# B&R Automation Studio project TD52 (part 124)

#### ChCCyclic.st
```iecst
(*******************************************************************************
ChC 			charge cooler

This code is confidential AND proprietary to the INNIO Company.
It may NOT be used in any form, OR reproduced in any manner,
without written permission of the INNIO Company.
Copyright, INNIO Company, 2019

Customized modifications: -
------------------------

History:
-------
V2.30	24.01.2008	LH			erstellt (Kopie von kv_schr)
 		06.02.2008	LH			angepasst an Auto-Tune Regler
V3.10.0	17.02.2010	lettenb.	corr.demand fan stage 1,2  step10: AND NOT FA_PLUS.Q --> AND FA_PLUS.Q
								corr. Anz_GK_anfhbt LIMIT(1->0,...)  	fehlerbehebung(robert mayer)
V3.99.0	21.02.2013	lettenb.	parts from pb3 included
		24.06.2013	lettenb.	xGRMin_Ventpos: Hy:= 1->0.01, bugfix
V4.00.0	03.03.2015	lettenb.	GK_frg (IN_HC.bChC_Rel) moved TO MM_CU
V4.03.0 07.08.2015  Denk		Manual operating auxiliaries control functionality added
        30.09.2015  Plattner	charge cooling pre heating OUT_HC.tChC_Heating.Do added
V4.07.0	09.08.2018	Schmid		2nd low temperature charge cooling circuit added
		08.01.2019	Schmid		redundant pump control
		22.02.2019	Schmid		Charge cooler heating bugfix

Instructions for use:
--------------------

Outstandings:
------------
(*******************************************************************************)
PROGRAM _CYCLIC
	//parameter definitions see settingsInit.st
	(* charge cooler 1st LT cooling circuit *)
	GK_var 			:= INT_TO_USINT(LIMIT(0, Para.iChC_OpMode,    2));		(* cooler mode (0-2)
																			0 = no cooler
																			1 = cooler level dependent on valve position supply water temperature controller
																			2 = cooler level dependent on charge (supply water) temperature *)
	GK_anz			:= INT_TO_USINT(LIMIT(1, Para.iChC_NumStages, 16));		(* number stages total (1-16)*)
	Anz_GK_anfhbt	:= INT_TO_USINT(LIMIT(0, Para.iChC_NumDemAux, GK_anz));	(* number stages with demand auxiliaries (0-16)*)
	GK_reg			:= INT_TO_USINT(LIMIT(1, Para.iChC_CtrNum, 9));			(* number controller for y for 3-way valve (1-9) (mode 1) *)
																			(* 1-8 = Ctr_Cust	plant controller - custom		*)
																			(*   9 = Ctr_ChC	charge temperature (t2') controller	*)

	(* charge cooler 2nd LT cooling circuit *)
	GK2_var 		:= INT_TO_USINT(LIMIT(0, Para.iChC2_OpMode,    22));	 (* cooler 2 fan operation mode (0-22)
																			 0	= LT circuits are connected, cooler fan controlled by 1st circuit (t2'), cooler 2 fan not connected
																			 11	= separate LT circuits, combi-cooler, cooler fan stage control for 2nd circuit dependent
																				  on temperature-control-valve position, cooler 2 fan not connected
																			 12	= separate LT circuits, combi-cooler, cooler fan stage control FOR 2nd circuit dependent
																				  on charge temperature (T1-HP), cooler 2 fan not connected
																			 21 = separate LT circuits, separate cooler fans, stage control dependent
																				  on temperature-control-valve position
																			 22 = separate LT circuits, separate cooler fans, stage control dependent
																				  on charge temperature (T1-HP) *)
	IF GK2_var > 20 THEN	(* separate 2nd charge cooler *)
		GK2_anz			:= INT_TO_USINT(LIMIT(1, Para.iChC2_NumStages, 16));	 	(* number stages total (1-16)*)
		Anz_GK2_anfhbt	:= INT_TO_USINT(LIMIT(0, Para.iChC2_NumDemAux, GK2_anz));	(* number stages with demand auxiliaries (0-16)*)
	ELSE					(* no 2nd charge cooler or combi-cooler *)
		GK2_anz			:= GK_anz;
		Anz_GK2_anfhbt	:= Anz_GK_anfhbt;
	END_IF;
	GK2_reg			:= INT_TO_USINT(LIMIT(1, Para.iChC2_CtrNum, 34));		 (* number controller for y for 3-way valve (1-8, 34)*)
																			 (* 1-8 = Ctr_Cust		plant controller - custom		*)
																			 (*  34 = Ctr_ChC_T1HP	charge temperature before high-pressure turbo charger (T1-HP) controller	*)

	(*------------------------------------------------------------------------------------------*)
	(* charge cooler pump *)
	OUT_HC.tChC_DemPump.Do		:= IN_HC.bEng_Aux_Dem_CDR
								OR IN_HC.tManAuxCtr.bChC_DemPump;	(* Manual operating auxiliaries control - Handbedienebene *)
	OUT_HC.bCCWP_Dem			:= OUT_HC.tChC_DemPump.Do;

	(* charge cooler 2 pump *)
	OUT_HC.tChC2_DemPump.Do		:= IN_HC.bEng_Aux_Dem_CDR
								OR IN_HC.tManAuxCtr.bChC2_DemPump;	(* Manual operating auxiliaries control - Handbedienebene *)
	OUT_HC.bCC2WP_Dem			:= OUT_HC.tChC2_DemPump.Do;

	(* release charge cooler from monitoring (remove not applicable parts) *)
	IN_HC.bChC_Rel;
	IN_HC.bChC2_Rel;

	(*==========================================================================================*)
	(* charge cooler control - stepper version *)
	IF GK_var > 0 THEN
		(* cooler stages ON/OFF according charge cooler mode *)
		(* if necessary change with limit value charge cooler water temperature *)
		bChC_Up   :=     bT_Ch_Hi2;
		bChC_Down := NOT bT_Ch_Hi1;

		(*------------------------------------------------------------------------------------------*)
		IF GK_var > 1 THEN
			Temp_KuehlerAustritt := 1;
		ELSE
			Temp_KuehlerAustritt := 0;
		END_IF;

		GK_vent			:=	0;
		GK_temp			:=	0;
		IF Temp_KuehlerAustritt THEN
			GK_temp		:=	1;
		ELSIF Para.bCtr_ChC THEN
			GK_vent		:=	1;
		END_IF;

		IF	Anz_GK_anfhbt > 0 THEN
			GK_anfhbt	:=	1;
		ELSE
			GK_anfhbt	:=	0;
		END_IF;

		FOR	i:=	1 TO 16 BY 1 DO
			gk_anfhbt[i] :=	0;
		END_FOR;
		FOR	i:=	1 TO Anz_GK_anfhbt BY 1	DO
			gk_anfhbt[i] :=	1;
		END_FOR;

		(* number stages effective *)
		Anz_GK_st		:=	MIN(GK_anz - (MAX(Anz_GK_anfhbt, 1) - 1), 16);

		zw := 1;
		FOR i:=	1 TO Anz_GK_st BY 1	DO
			zw := zw * 2;
		END_FOR;

		FA_INIT_1.Word	:=	UDINT_TO_UINT(zw - 1);
		FA_INIT_1;
		ST_1			:=	FA_INIT_1.Bit00;
		ST_2			:=	FA_INIT_1.Bit01;
		ST_3			:=	FA_INIT_1.Bit02;
		ST_4			:=	FA_INIT_1.Bit03;
		ST_5			:=	FA_INIT_1.Bit04;
		ST_6			:=	FA_INIT_1.Bit05;
		ST_7			:=	FA_INIT_1.Bit06;
		ST_8			:=	FA_INIT_1.Bit07;
		ST_9			:=	FA_INIT_1.Bit08;
		ST_10			:=	FA_INIT_1.Bit09;
		ST_11			:=	FA_INIT_1.Bit10;
		ST_12			:=	FA_INIT_1.Bit11;
		ST_13			:=	FA_INIT_1.Bit12;
		ST_14			:=	FA_INIT_1.Bit13;
		ST_15			:=	FA_INIT_1.Bit14;
		ST_16			:=	FA_INIT_1.Bit15;

		(* activation cooler stages *)
		Anz_GK_vent		:=	MIN(GK_anz, 16);

		zw := 1;
		FOR	i:=	1 TO Anz_GK_vent BY 1 DO
			zw := zw * 2;
		END_FOR;

		FA_INIT_2.Word	:=	UDINT_TO_UINT(zw - 1);
		FA_INIT_2;
		GK_ST_1			:=	FA_INIT_2.Bit00;
		GK_ST_2			:=	FA_INIT_2.Bit01;
		GK_ST_3			:=	FA_INIT_2.Bit02;
		GK_ST_4			:=	FA_INIT_2.Bit03;
		GK_ST_5			:=	FA_INIT_2.Bit04;
		GK_ST_6			:=	FA_INIT_2.Bit05;
		GK_ST_7			:=	FA_INIT_2.Bit06;
		GK_ST_8			:=	FA_INIT_2.Bit07;
		GK_ST_9			:=	FA_INIT_2.Bit08;
		GK_ST_10		:=	FA_INIT_2.Bit09;
		GK_ST_11		:=	FA_INIT_2.Bit10;
		GK_ST_12		:=	FA_INIT_2.Bit11;
		GK_ST_13		:=	FA_INIT_2.Bit12;
		GK_ST_14		:=	FA_INIT_2.Bit13;
		GK_ST_15		:=	FA_INIT_2.Bit14;
		GK_ST_16		:=	FA_INIT_2.Bit15;

	//	(* 3-way cooler valve *)
		CASE GK_reg OF										(* selection plant ctr # for 3-way valve (1-11) (cooler mode 1/3) *)
			1:	F_SPSR		:=	IN_HC.tCtr_Cust1_In.enable;	(* 1-8 = custom plant ctr - device temperature *)
				rValvePos	:=	IN_HC.tCtr_Cust1_Out.Y;
				REG_INVERT	:=	Para.tCtr_Cust1.invert;
			2:	F_SPSR		:=	IN_HC.tCtr_Cust2_In.enable;
				rValvePos	:=	IN_HC.tCtr_Cust2_Out.Y;
				REG_INVERT	:=	Para.tCtr_Cust2.invert;
			3:	F_SPSR		:=	IN_HC.tCtr_Cust3_In.enable;
				rValvePos	:=	IN_HC.tCtr_Cust3_Out.Y;
				REG_INVERT	:=	Para.tCtr_Cust3.invert;
			4:	F_SPSR		:=	IN_HC.tCtr_Cust4_In.enable;
				rValvePos	:=	IN_HC.tCtr_Cust4_Out.Y;
				REG_INVERT	:=	Para.tCtr_Cust4.invert;
			5:	F_SPSR		:=	IN_HC.tCtr_Cust5_In.enable;
				rValvePos	:=	IN_HC.tCtr_Cust5_Out.Y;
				REG_INVERT	:=	Para.tCtr_Cust5.invert;
			6:	F_SPSR		:=	IN_HC.tCtr_Cust6_In.enable;
				rValvePos	:=	IN_HC.tCtr_Cust6_Out.Y;
				REG_INVERT	:=	Para.tCtr_Cust6.invert;
			7:	F_SPSR		:=	IN_HC.tCtr_Cust7_In.enable;
				rValvePos	:=	IN_HC.tCtr_Cust7_Out.Y;
				REG_INVERT	:=	Para.tCtr_Cust7.invert;
			8:	F_SPSR		:=	IN_HC.tCtr_Cust8_In.enable;
				rValvePos	:=	IN_HC.tCtr_Cust8_Out.Y;
				REG_INVERT	:=	Para.tCtr_Cust8.invert;
			9:	F_SPSR		:=	tCtr_ChC_In.enable;			(* 9   = charge temperature controller *)
				rValvePos	:=	tCtr_ChC_Out.Y;
				REG_INVERT	:=	Para.tCtr_ChC.invert;
			ELSE
				F_SPSR		:=	FALSE;
				rValvePos	:=	0.0;
				REG_INVERT	:=	FALSE;
		END_CASE;

		IF	NOT REG_INVERT	THEN
			rValvePos	:=	1.0 - rValvePos;
		END_IF;

	    (*---------------------------------------------------------------------------*)
		(* cooler ON *)
		xGRMax_Ventpos(Gw:= Para.rChC_ValPosLimHi_On, Hy:= Para.rChC_ValPosHyHi_On, In:= rValvePos);

		xTOF_GK_AUS.IN	:=	GK_vent AND xGRMax_Ventpos.Q AND IN_HC.tPB2MM.bParaSetupOk AND USINT_TO_BOOL(F_SPSR) OR
							GK_temp AND ((bChC_Up OR GK_EIN AND NOT bChC_Down) OR GK_EIN AND M_GKV2);
		xTOF_GK_AUS.PT 	:=  Para.tiChC_DelayOff;
	    xTOF_GK_AUS();

	    GK_EIN			:=	(xTOF_GK_AUS.Q OR GK_anfhbt) AND IN_HC.bEng_Aux_Dem_CDR AND IN_HC.bChC_Rel;

	    (*---------------------------------------------------------------------------*)
		(* cooler stages plus *)
		xGRMax_Ventpos2(Gw:= Para.rChC_ValPosLimStageUp, Hy:= 0.01, In:= rValvePos);

		GK_PLUS			:= (GK_vent AND xGRMax_Ventpos2.Q AND IN_HC.tPB2MM.bParaSetupOk)
						OR (GK_temp AND bChC_Up);

	    (*---------------------------------------------------------------------------*)
		(* cooler stages minus *)
		xGRMin_Ventpos(Gw := Para.rChC_ValPosLimStageDown, Hy := 0.01, In := rValvePos);

		GK_MINUS		:=((xGRMin_Ventpos.Q AND IN_HC.tPB2MM.bParaSetupOk AND GK_vent) OR (GK_temp AND bChC_Down))
					AND NOT GK_PLUS;

	    (*---------------------------------------------------------------------------*)
		(* delay between stages ON *)
		xTOF_PLUS(IN:= plus, PT:= Para.tiChC_DelayStageUp);
		xR_TRIG_PLUS(CLK:= GK_PLUS AND NOT xTOF_PLUS.Q);

	    (*---------------------------------------------------------------------------*)
		(* delay between stages OFF *)
		xTOF_MINUS(IN:= minus, PT:= Para.tiChC_DelayStageDown);
		xR_TRIG_MINUS(CLK:=	GK_MINUS AND NOT xTOF_MINUS.Q);

	    (*---------------------------------------------------------------------------*)
		(* reset stage maschine *)
		IF	NOT GK_EIN	THEN
			schritt	:=	0;
		END_IF;

		(* state maschine *)
		CASE schritt OF	00:	(* cooler stopped *)
			FA_INIT_3.Word	:=	0;
			FA_INIT_3;
			M_GKV1			:=	FA_INIT_3.Bit00;
			M_GKV2			:=	FA_INIT_3.Bit01;
			M_GKV3			:=	FA_INIT_3.Bit02;
			M_GKV4			:=	FA_INIT_3.Bit03;
			M_GKV5			:=	FA_INIT_3.Bit04;
			M_GKV6			:=	FA_INIT_3.Bit05;
			M_GKV7			:=	FA_INIT_3.Bit06;
			M_GKV8			:=	FA_INIT_3.Bit07;
			M_GKV9			:=	FA_INIT_3.Bit08;
			M_GKV10			:=	FA_INIT_3.Bit09;
			M_GKV11			:=	FA_INIT_3.Bit10;
			M_GKV12			:=	FA_INIT_3.Bit11;
			M_GKV13			:=	FA_INIT_3.Bit12;
			M_GKV14			:=	FA_INIT_3.Bit13;
			M_GKV15			:=	FA_INIT_3.Bit14;
			M_GKV16			:=	FA_INIT_3.Bit15;

			(* ON 1.stage *)
			IF	GK_EIN	THEN
				schritt		:=	10;
			END_IF;

		10:	(* cooler stage 1 *)
			M_GKV1			:=	1;
			M_GKV2			:=	0;
			(* ON 2.stage *)
			IF	GK_PLUS AND(   (GK_temp AND bChC_Up AND xR_TRIG_PLUS.Q)
				            OR (GK_vent AND xGRMax_Ventpos2.Q)) THEN
				schritt		:=	20;
			END_IF;

		20:	(* cooler stage 2 *)
			M_GKV2			:=	1;
			M_GKV3			:=	0;
			(* ON 3.stage *)
			IF	GK_PLUS AND xR_TRIG_PLUS.Q AND ST_3	THEN
				schritt		:=	30;
			END_IF;
			(* OFF 3.stage *)
			IF	GK_MINUS AND (xR_TRIG_MINUS.Q OR NOT ST_3) THEN
				schritt		:=	10;
			END_IF;

		30:	(* cooler stage 3 *)
			M_GKV3			:=	1;
			M_GKV4			:=	0;
			(* ON 4.stage *)
			IF	GK_PLUS AND xR_TRIG_PLUS.Q AND ST_4	THEN
				schritt		:=	40;
			END_IF;
			(* OFF 3.stage *)
			IF	GK_MINUS AND (xR_TRIG_MINUS.Q OR NOT ST_4)	THEN
				schritt		:=	20;
			END_IF;

		40:	(* cooler stage 4 *)
			M_GKV4			:=	1;
			M_GKV5			:=	0;
			(* ON 5.stage *)
			IF	GK_PLUS AND xR_TRIG_PLUS.Q AND ST_5	THEN
				schritt		:=	50;
			END_IF;
			(* OFF 4.stage *)
			IF	GK_MINUS AND (xR_TRIG_MINUS.Q OR NOT ST_5) THEN
				schritt		:=	30;
			END_IF;

		50:	(* cooler stage 5 *)
			M_GKV5			:=	1;
			M_GKV6			:=	0;
			(* ON 6.stage *)
			IF	GK_PLUS AND xR_TRIG_PLUS.Q AND ST_6	THEN
				schritt		:=	60;
			END_IF;
			(* OFF 5.stage *)
			IF	GK_MINUS AND (xR_TRIG_MINUS.Q OR NOT ST_6) THEN
				schritt		:=	40;
			END_IF;

		60:	(* cooler stage 6 *)
			M_GKV6			:=	1;
			M_GKV7			:=	0;
			(* ON 7.stage *)
			IF	GK_PLUS AND xR_TRIG_PLUS.Q AND ST_7	THEN
				schritt		:=	70;
			END_IF;
			(* OFF 6.stage *)
			IF	GK_MINUS AND (xR_TRIG_MINUS.Q OR NOT ST_7) THEN
				schritt		:=	50;
			END_IF;

		70:	(* cooler stage 7 *)
			M_GKV7			:=	1;
			M_GKV8			:=	0;
			(* ON 8.stage *)
			IF	GK_PLUS AND xR_TRIG_PLUS.Q AND ST_8	THEN
				schritt		:=	80;
			END_IF;
			(* OFF 7.stage *)
			IF	GK_MINUS AND (xR_TRIG_MINUS.Q OR NOT ST_8) THEN
				schritt		:=	60;
			END_IF;

		80:	(* cooler stage 8 *)
			M_GKV8			:=	1;
			M_GKV9			:=	0;
			(* ON 9.stage *)
			IF	GK_PLUS AND xR_TRIG_PLUS.Q AND ST_9	THEN
				schritt		:=	90;
			END_IF;
			(* OFF 8.stage *)
			IF	GK_MINUS AND (xR_TRIG_MINUS.Q OR NOT ST_9) THEN
				schritt		:=	70;
			END_IF;

		90:	(* cooler stage 9 *)
			M_GKV9			:=	1;
			M_GKV10			:=	0;
			(* ON 10.stage *)
			IF	GK_PLUS AND xR_TRIG_PLUS.Q AND ST_10 THEN
				schritt		:=	100;
			END_IF;
			(* OFF 9.stage *)
			IF	GK_MINUS AND (xR_TRIG_MINUS.Q OR NOT ST_10)	THEN
				schritt		:=	80;
			END_IF;

		100:(* cooler stage 10 *)
			M_GKV10			:=	1;
			M_GKV11			:=	0;
			(* ON 11.stage *)
			IF	GK_PLUS AND xR_TRIG_PLUS.Q AND ST_11 THEN
				schritt		:=	110;
			END_IF;
			(* OFF 10.stage *)
			IF	GK_MINUS AND (xR_TRIG_MINUS.Q OR NOT ST_11)	THEN
				schritt		:=	90;
			END_IF;

		110:(* cooler stage 11 *)
			M_GKV11			:=	1;
			M_GKV12			:=	0;
			(* ON 12.stage *)
			IF	GK_PLUS AND xR_TRIG_PLUS.Q AND ST_12 THEN
				schritt		:=	120;
			END_IF;
			(* OFF 11.stage *)
			IF	GK_MINUS AND (xR_TRIG_MINUS.Q OR NOT ST_12)	THEN
				schritt		:=	100;
			END_IF;

		120:(* cooler stage 12 *)
			M_GKV12			:=	1;
			M_GKV13			:=	0;
			(* ON 13.stage *)
			IF	GK_PLUS AND xR_TRIG_PLUS.Q AND ST_13 THEN
				schritt		:=	130;
			END_IF;
			(* OFF 12.stage *)
			IF	GK_MINUS AND (xR_TRIG_MINUS.Q OR NOT ST_13)	THEN
				schritt		:=	110;
			END_IF;

		130:(* cooler stage 13 *)
			M_GKV13			:=	1;
			M_GKV14			:=	0;
			(* ON 14.stage *)
			IF	GK_PLUS AND xR_TRIG_PLUS.Q AND ST_14 THEN
				schritt		:=	140;
			END_IF;
			(* OFF 13.stage *)
			IF	GK_MINUS AND (xR_TRIG_MINUS.Q OR NOT ST_14)	THEN
				schritt		:=	120;
			END_IF;

		140:(* cooler stage 14 *)
			M_GKV14			:=	1;
			M_GKV15			:=	0;
			(* ON 15.stage *)
			IF	GK_PLUS AND xR_TRIG_PLUS.Q AND ST_15 THEN
				schritt		:=	150;
			END_IF;
			(* OFF 14.stage *)
			IF	GK_MINUS AND (xR_TRIG_MINUS.Q OR NOT ST_15)	THEN
				schritt		:=	130;
			END_IF;

		150:(* cooler stage 15 *)
			M_GKV15			:=	1;
			M_GKV16			:=	0;
			(* ON 16.stage *)
			IF	GK_PLUS AND xR_TRIG_PLUS.Q AND ST_16 THEN
				schritt		:=	160;
			END_IF;
			(* OFF 15.stage *)
			IF	GK_MINUS AND (xR_TRIG_MINUS.Q OR NOT ST_16)	THEN
				schritt		:=	140;
			END_IF;

		160:(* cooler stage 16 *)
			M_GKV16			:=	1;
			(* OFF 16.stage *)
			IF	GK_MINUS THEN
				schritt		:=	150;
			END_IF;
		END_CASE;

		(* charge cooler pump
		GKP_EIN				:=	M_GKV1; *)

		(* connection cooler stages to sequencing *)
		GK_ST1		:=	M_GKV1;

		GK_ST2		:=	M_GKV1 AND gk_anfhbt[2] OR
						M_GKV2;

		GK_ST3		:=	M_GKV1 AND gk_anfhbt[3] OR
						M_GKV2 AND gk_anfhbt[2] OR
						M_GKV3;

		GK_ST4		:=	M_GKV1 AND gk_anfhbt[4] OR
						M_GKV2 AND gk_anfhbt[3] OR
						M_GKV3 AND gk_anfhbt[2] OR
						M_GKV4;

		GK_ST5		:=	M_GKV1 AND gk_anfhbt[5] OR
						M_GKV2 AND gk_anfhbt[4] OR
						M_GKV3 AND gk_anfhbt[3] OR
						M_GKV4 AND gk_anfhbt[2] OR
						M_GKV5;

		GK_ST6		:=	M_GKV1 AND gk_anfhbt[6] OR
						M_GKV2 AND gk_anfhbt[5] OR
						M_GKV3 AND gk_anfhbt[4] OR
						M_GKV4 AND gk_anfhbt[3] OR
						M_GKV5 AND gk_anfhbt[2] OR
						M_GKV6;

		GK_ST7		:=	M_GKV1 AND gk_anfhbt[7] OR
						M_GKV2 AND gk_anfhbt[6] OR
						M_GKV3 AND gk_anfhbt[5] OR
						M_GKV4 AND gk_anfhbt[4] OR
						M_GKV5 AND gk_anfhbt[3] OR
						M_GKV6 AND gk_anfhbt[2] OR
						M_GKV7;

		GK_ST8		:=	M_GKV1 AND gk_anfhbt[8] OR
						M_GKV2 AND gk_anfhbt[7] OR
						M_GKV3 AND gk_anfhbt[6] OR
						M_GKV4 AND gk_anfhbt[5] OR
						M_GKV5 AND gk_anfhbt[4] OR
						M_GKV6 AND gk_anfhbt[3] OR
						M_GKV7 AND gk_anfhbt[2] OR
						M_GKV8;

		GK_ST9		:=	M_GKV1 AND gk_anfhbt[9] OR
						M_GKV2 AND gk_anfhbt[8] OR
						M_GKV3 AND gk_anfhbt[7] OR
						M_GKV4 AND gk_anfhbt[6] OR
						M_GKV5 AND gk_anfhbt[5] OR
						M_GKV6 AND gk_anfhbt[4] OR
						M_GKV7 AND gk_anfhbt[3] OR
						M_GKV8 AND gk_anfhbt[2] OR
						M_GKV9;

		GK_ST10		:=	M_GKV1 AND gk_anfhbt[10] OR
						M_GKV2 AND gk_anfhbt[9]  OR
						M_GKV3 AND gk_anfhbt[8]  OR
						M_GKV4 AND gk_anfhbt[7]  OR
						M_GKV5 AND gk_anfhbt[6]  OR
						M_GKV6 AND gk_anfhbt[5]  OR
						M_GKV7 AND gk_anfhbt[4]  OR
						M_GKV8 AND gk_anfhbt[3]  OR
						M_GKV9 AND gk_anfhbt[2]  OR
						M_GKV10;

		GK_ST11		:=	M_GKV1  AND gk_anfhbt[11] OR
						M_GKV2  AND gk_anfhbt[10] OR
						M_GKV3  AND gk_anfhbt[9]  OR
						M_GKV4  AND gk_anfhbt[8]  OR
						M_GKV5  AND gk_anfhbt[7]  OR
						M_GKV6  AND gk_anfhbt[6]  OR
						M_GKV7  AND gk_anfhbt[5]  OR
						M_GKV8  AND gk_anfhbt[4]  OR
						M_GKV9  AND gk_anfhbt[3]  OR
						M_GKV10 AND gk_anfhbt[2]  OR
						M_GKV11;

		GK_ST12		:=	M_GKV1  AND gk_anfhbt[12] OR
						M_GKV2  AND gk_anfhbt[11] OR
						M_GKV3  AND gk_anfhbt[10] OR
						M_GKV4  AND gk_anfhbt[9]  OR
						M_GKV5  AND gk_anfhbt[8]  OR
						M_GKV6  AND gk_anfhbt[7]  OR
						M_GKV7  AND gk_anfhbt[6]  OR
						M_GKV8  AND gk_anfhbt[5]  OR
						M_GKV9  AND gk_anfhbt[4]  OR
						M_GKV10 AND gk_anfhbt[3]  OR
						M_GKV11 AND gk_anfhbt[2]  OR
						M_GKV12;

		GK_ST13		:=	M_GKV1  AND gk_anfhbt[13] OR
						M_GKV2  AND gk_anfhbt[12] OR
						M_GKV3  AND gk_anfhbt[11] OR
						M_GKV4  AND gk_anfhbt[10] OR
						M_GKV5  AND gk_anfhbt[9]  OR
						M_GKV6  AND gk_anfhbt[8]  OR
						M_GKV7  AND gk_anfhbt[7]  OR
						M_GKV8  AND gk_anfhbt[6]  OR
						M_GKV9  AND gk_anfhbt[5]  OR
						M_GKV10 AND gk_anfhbt[4]  OR
						M_GKV11 AND gk_anfhbt[3]  OR
						M_GKV12 AND gk_anfhbt[2]  OR
						M_GKV13;

		GK_ST14		:=	M_GKV1  AND gk_anfhbt[14] OR
						M_GKV2  AND gk_anfhbt[13] OR
						M_GKV3  AND gk_anfhbt[12] OR
						M_GKV4  AND gk_anfhbt[11] OR
						M_GKV5  AND gk_anfhbt[10] OR
						M_GKV6  AND gk_anfhbt[9]  OR
						M_GKV7  AND gk_anfhbt[8]  OR
						M_GKV8  AND gk_anfhbt[7]  OR
						M_GKV9  AND gk_anfhbt[6]  OR
						M_GKV10 AND gk_anfhbt[5]  OR
						M_GKV11 AND gk_anfhbt[4]  OR
						M_GKV12 AND gk_anfhbt[3]  OR
						M_GKV13 AND gk_anfhbt[2]  OR
						M_GKV14;

		GK_ST15		:=	M_GKV1  AND gk_anfhbt[15] OR
						M_GKV2  AND gk_anfhbt[14] OR
						M_GKV3  AND gk_anfhbt[13] OR
						M_GKV4  AND gk_anfhbt[12] OR
						M_GKV5  AND gk_anfhbt[11] OR
						M_GKV6  AND gk_anfhbt[10] OR
						M_GKV7  AND gk_anfhbt[9]  OR
						M_GKV8  AND gk_anfhbt[8]  OR
						M_GKV9  AND gk_anfhbt[7]  OR
						M_GKV10 AND gk_anfhbt[6]  OR
						M_GKV11 AND gk_anfhbt[5]  OR
						M_GKV12 AND gk_anfhbt[4]  OR
						M_GKV13 AND gk_anfhbt[3]  OR
						M_GKV14 AND gk_anfhbt[2]  OR
						M_GKV15;

		GK_ST16		:=	M_GKV1  AND gk_anfhbt[16] OR
						M_GKV2  AND gk_anfhbt[15] OR
						M_GKV3  AND gk_anfhbt[14] OR
						M_GKV4  AND gk_anfhbt[13] OR
						M_GKV5  AND gk_anfhbt[12] OR
						M_GKV6  AND gk_anfhbt[11] OR
						M_GKV7  AND gk_anfhbt[10] OR
						M_GKV8  AND gk_anfhbt[9]  OR
						M_GKV9  AND gk_anfhbt[8]  OR
						M_GKV10 AND gk_anfhbt[7]  OR
						M_GKV11 AND gk_anfhbt[6]  OR
						M_GKV12 AND gk_anfhbt[5]  OR
						M_GKV13 AND gk_anfhbt[4]  OR
						M_GKV14 AND gk_anfhbt[3]  OR
						M_GKV15 AND gk_anfhbt[2]  OR
						M_GKV16;

		(* copy for summation *)
		GKST[1]		:=	BOOL_TO_USINT(M_GKV1);
		GKST[2]		:=	BOOL_TO_USINT(M_GKV2);
		GKST[3]		:=	BOOL_TO_USINT(M_GKV3);
		GKST[4]		:=	BOOL_TO_USINT(M_GKV4);
		GKST[5]		:=	BOOL_TO_USINT(M_GKV5);
		GKST[6]		:=	BOOL_TO_USINT(M_GKV6);
		GKST[7]		:=	BOOL_TO_USINT(M_GKV7);
		GKST[8]		:=	BOOL_TO_USINT(M_GKV8);
		GKST[9]		:=	BOOL_TO_USINT(M_GKV9);
		GKST[10]	:=	BOOL_TO_USINT(M_GKV10);
		GKST[11]	:=	BOOL_TO_USINT(M_GKV11);
		GKST[12]	:=	BOOL_TO_USINT(M_GKV12);
		GKST[13]	:=	BOOL_TO_USINT(M_GKV13);
		GKST[14]	:=	BOOL_TO_USINT(M_GKV14);
		GKST[15]	:=	BOOL_TO_USINT(M_GKV15);
		GKST[16]	:=	BOOL_TO_USINT(M_GKV16);

		(* ON/OFF coolerstage *)
		summe := 0;
		FOR i:=	1 TO 16 BY 1 DO
			summe := summe + GKST[i];
		END_FOR;

		plus :=	0;
		IF summe > summe_old THEN
			plus := 1;
		END_IF;

		minus := 0;
		IF summe < summe_old THEN
			minus := 1;
		END_IF;

		summe_old := summe;

	END_IF;

	(*==========================================================================================*)
	(* charge cooler 2 control - stepper version *)
	IF GK2_var > 0 THEN
		(* cooler stages ON/OFF according charge cooler 2 mode *)
		(* if necessary change with limit value charge cooler 2 water temperature *)
		bChC2_Up   :=     bT_Ch2_Hi2;
		bChC2_Down := NOT bT_Ch2_Hi1;

		(*------------------------------------------------------------------------------------------*)
		(* charge cooler 2 stage control mode *)
		GK2_vent			:=	0;
		GK2_temp			:=	0;
		IF (GK2_var MOD 10) = 2 THEN	(* via charge temperature T1-HP limits *)
			GK2_temp		:=	1;
		ELSIF (GK2_var MOD 10) = 1 AND Para.bCtr_ChC_T1HP THEN	(* via temperature-control-valve position *)
			GK2_vent		:=	1;
		END_IF;

		IF	Anz_GK2_anfhbt > 0 THEN
			GK2_anfhbt	:=	1;
		ELSE
			GK2_anfhbt	:=	0;
		END_IF;

		FOR	i:=	1 TO 16 DO
			IF i <= Anz_GK2_anfhbt THEN
				gk2_anfhbt[i] :=	1;
			ELSE
				gk2_anfhbt[i] :=	0;
			END_IF;
		END_FOR;

		(* number stages effective - charge cooler 2*)
		Anz_GK2_st		:=	MIN(GK2_anz - (MAX(Anz_GK2_anfhbt, 1) - 1), 16);

		zw := 1;
		FOR i:=	1 TO Anz_GK2_st BY 1	DO
			zw := zw * 2;
		END_FOR;

		FA2_INIT_1.Word	:=	UDINT_TO_UINT(zw - 1);
		FA2_INIT_1;
		ST2_1			:=	FA2_INIT_1.Bit00;
		ST2_2			:=	FA2_INIT_1.Bit01;
		ST2_3			:=	FA2_INIT_1.Bit02;
		ST2_4			:=	FA2_INIT_1.Bit03;
		ST2_5			:=	FA2_INIT_1.Bit04;
		ST2_6			:=	FA2_INIT_1.Bit05;
		ST2_7			:=	FA2_INIT_1.Bit06;
		ST2_8			:=	FA2_INIT_1.Bit07;
		ST2_9			:=	FA2_INIT_1.Bit08;
		ST2_10			:=	FA2_INIT_1.Bit09;
		ST2_11			:=	FA2_INIT_1.Bit10;
		ST2_12			:=	FA2_INIT_1.Bit11;
		ST2_13			:=	FA2_INIT_1.Bit12;
		ST2_14			:=	FA2_INIT_1.Bit13;
		ST2_15			:=	FA2_INIT_1.Bit14;
		ST2_16			:=	FA2_INIT_1.Bit15;

		(* enable cooler stages - charge cooler 2 *)
		Anz_GK2_vent		:=	MIN(GK2_anz, 16);

		zw := 1;
		FOR	i:=	1 TO Anz_GK2_vent BY 1 DO
			zw := zw * 2;
		END_FOR;

		FA2_INIT_2.Word	:=	UDINT_TO_UINT(zw - 1);
		FA2_INIT_2;
		GK2_ST_1			:=	FA2_INIT_2.Bit00;
		GK2_ST_2			:=	FA2_INIT_2.Bit01;
		GK2_ST_3			:=	FA2_INIT_2.Bit02;
		GK2_ST_4			:=	FA2_INIT_2.Bit03;
		GK2_ST_5			:=	FA2_INIT_2.Bit04;
		GK2_ST_6			:=	FA2_INIT_2.Bit05;
		GK2_ST_7			:=	FA2_INIT_2.Bit06;
		GK2_ST_8			:=	FA2_INIT_2.Bit07;
		GK2_ST_9			:=	FA2_INIT_2.Bit08;
		GK2_ST_10			:=	FA2_INIT_2.Bit09;
		GK2_ST_11			:=	FA2_INIT_2.Bit10;
		GK2_ST_12			:=	FA2_INIT_2.Bit11;
		GK2_ST_13			:=	FA2_INIT_2.Bit12;
		GK2_ST_14			:=	FA2_INIT_2.Bit13;
		GK2_ST_15			:=	FA2_INIT_2.Bit14;
		GK2_ST_16			:=	FA2_INIT_2.Bit15;

	//	(* 3-way cooler valve - charge cooler 2 *)
		CASE GK2_reg OF										(* selection plant ctr # for 3-way valve (1-11) (cooler mode 1/3) *)
			1:	F2_SPSR		:=	IN_HC.tCtr_Cust1_In.enable;	(* 1-8 = custom plant ctr - device temperature *)
				rValvePos2	:=	IN_HC.tCtr_Cust1_Out.Y;
				REG2_INVERT	:=	Para.tCtr_Cust1.invert;
			2:	F2_SPSR		:=	IN_HC.tCtr_Cust2_In.enable;
				rValvePos2	:=	IN_HC.tCtr_Cust2_Out.Y;
				REG2_INVERT	:=	Para.tCtr_Cust2.invert;
			3:	F2_SPSR		:=	IN_HC.tCtr_Cust3_In.enable;
				rValvePos2	:=	IN_HC.tCtr_Cust3_Out.Y;
				REG2_INVERT	:=	Para.tCtr_Cust3.invert;
			4:	F2_SPSR		:=	IN_HC.tCtr_Cust4_In.enable;
				rValvePos2	:=	IN_HC.tCtr_Cust4_Out.Y;
				REG2_INVERT	:=	Para.tCtr_Cust4.invert;
			5:	F2_SPSR		:=	IN_HC.tCtr_Cust5_In.enable;
				rValvePos2	:=	IN_HC.tCtr_Cust5_Out.Y;
				REG2_INVERT	:=	Para.tCtr_Cust5.invert;
			6:	F2_SPSR		:=	IN_HC.tCtr_Cust6_In.enable;
				rValvePos2	:=	IN_HC.tCtr_Cust6_Out.Y;
				REG2_INVERT	:=	Para.tCtr_Cust6.invert;
			7:	F2_SPSR		:=	IN_HC.tCtr_Cust7_In.enable;
				rValvePos2	:=	IN_HC.tCtr_Cust7_Out.Y;
				REG2_INVERT	:=	Para.tCtr_Cust7.invert;
			8:	F2_SPSR		:=	IN_HC.tCtr_Cust8_In.enable;
				rValvePos2	:=	IN_HC.tCtr_Cust8_Out.Y;
				REG2_INVERT	:=	Para.tCtr_Cust8.invert;
			34:	F2_SPSR		:=	tCtr_ChC_T1HP_In.enable;		(* 34   = charge temperature before high-pressure turbo charger (T1HP) controller *)
				rValvePos2	:=	tCtr_ChC_T1HP_Out.Y;
				REG2_INVERT	:=	Para.tCtr_ChC_T1HP.invert;
			ELSE
				F2_SPSR		:=	FALSE;
				rValvePos2	:=	0.0;
				REG2_INVERT	:=	FALSE;
		END_CASE;

		IF	NOT REG2_INVERT	THEN
			rValvePos2	:=	1.0 - rValvePos2;
		END_IF;

	    (*---------------------------------------------------------------------------*)
		(* cooler 2 ON *)
		xGRMax2_Ventpos(Gw:= Para.rChC2_ValPosLimHi_On, Hy:= Para.rChC2_ValPosHyHi_On, In:= rValvePos2);

		xTOF_GK2_AUS.IN	:=	GK2_vent AND xGRMax2_Ventpos.Q AND IN_HC.tPB2MM.bParaSetupOk AND USINT_TO_BOOL(F2_SPSR) OR
							GK2_temp AND ((bChC2_Up OR GK2_EIN AND NOT bChC2_Down) OR GK2_EIN AND M_GK2V2);
		xTOF_GK2_AUS.PT :=  Para.tiChC2_DelayOff;
	    xTOF_GK2_AUS();

	    GK2_EIN			:=	(xTOF_GK2_AUS.Q OR GK2_anfhbt) AND IN_HC.bEng_Aux_Dem_CDR AND IN_HC.bChC2_Rel;

	    (*---------------------------------------------------------------------------*)
		(* cooler 2 stages plus *)
		xGRMax2_Ventpos2(Gw:= Para.rChC2_ValPosLimStageUp, Hy:= 0.01, In:= rValvePos2);

		GK2_PLUS		:= (GK2_vent AND xGRMax2_Ventpos2.Q AND IN_HC.tPB2MM.bParaSetupOk)
						OR (GK2_temp AND bChC2_Up);

	    (*---------------------------------------------------------------------------*)
		(* cooler 2 stages minus *)
		xGRMin2_Ventpos(Gw := Para.rChC2_ValPosLimStageDown, Hy := 0.01, In := rValvePos2);

		GK2_MINUS		:=((GK2_vent AND xGRMin2_Ventpos.Q AND IN_HC.tPB2MM.bParaSetupOk) OR (GK2_temp AND bChC2_Down))
					AND NOT GK2_PLUS;

	    (*---------------------------------------------------------------------------*)
		(* delay between stages ON - charge cooler 2 *)
		xTOF_PLUS2(IN:= plus2, PT:= Para.tiChC2_DelayStageUp);
		xR_TRIG_PLUS2(CLK:= GK2_PLUS AND NOT xTOF_PLUS2.Q);

	    (*---------------------------------------------------------------------------*)
		(* delay between stages OFF - charge cooler 2 *)
		xTOF_MINUS2(IN:= minus2, PT:= Para.tiChC2_DelayStageDown);
		xR_TRIG_MINUS2(CLK:= GK2_MINUS AND NOT xTOF_MINUS2.Q);

	    (*---------------------------------------------------------------------------*)
		(* reset stage maschine - charge cooler 2 *)
		IF	NOT GK2_EIN	THEN
			schritt2	:=	0;
		END_IF;

		(* stage maschine - charge cooler 2 *)
		CASE schritt2 OF 00:	(* cooler 2 stopped *)
			FA2_INIT_3.Word	:=	0;
			FA2_INIT_3;
			M_GK2V1			:=	FA2_INIT_3.Bit00;
			M_GK2V2			:=	FA2_INIT_3.Bit01;
			M_GK2V3			:=	FA2_INIT_3.Bit02;
			M_GK2V4			:=	FA2_INIT_3.Bit03;
			M_GK2V5			:=	FA2_INIT_3.Bit04;
			M_GK2V6			:=	FA2_INIT_3.Bit05;
			M_GK2V7			:=	FA2_INIT_3.Bit06;
			M_GK2V8			:=	FA2_INIT_3.Bit07;
			M_GK2V9			:=	FA2_INIT_3.Bit08;
			M_GK2V10		:=	FA2_INIT_3.Bit09;
			M_GK2V11		:=	FA2_INIT_3.Bit10;
			M_GK2V12		:=	FA2_INIT_3.Bit11;
			M_GK2V13		:=	FA2_INIT_3.Bit12;
			M_GK2V14		:=	FA2_INIT_3.Bit13;
			M_GK2V15		:=	FA2_INIT_3.Bit14;
			M_GK2V16		:=	FA2_INIT_3.Bit15;

			(* ON 1.stage *)
			IF	GK2_EIN	THEN
				schritt2	:=	10;
			END_IF;

		10:	(* cooler 2 stage 1 *)
			M_GK2V1			:=	1;
			M_GK2V2			:=	0;
			(* ON 2.stage *)
			IF	GK2_PLUS AND(   (GK2_temp AND bChC2_Up AND xR_TRIG_PLUS2.Q)
				            OR (GK2_vent AND xGRMax2_Ventpos2.Q)) THEN
				schritt2	:=	20;
			END_IF;

		20:	(* cooler 2 stage 2 *)
			M_GK2V2			:=	1;
			M_GK2V3			:=	0;
			(* ON 3.stage *)
			IF	GK2_PLUS AND xR_TRIG_PLUS2.Q AND ST2_3	THEN
				schritt2	:=	30;
			END_IF;
			(* OFF 3.stage *)
			IF	GK2_MINUS AND (xR_TRIG_MINUS2.Q OR NOT ST2_3) THEN
				schritt2	:=	10;
			END_IF;

		30:	(* cooler 2 stage 3 *)
			M_GK2V3			:=	1;
			M_GK2V4			:=	0;
			(* ON 4.stage *)
			IF	GK2_PLUS AND xR_TRIG_PLUS2.Q AND ST2_4	THEN
				schritt2	:=	40;
			END_IF;
			(* OFF 3.stage *)
			IF	GK2_MINUS AND (xR_TRIG_MINUS2.Q OR NOT ST2_4)	THEN
				schritt2	:=	20;
			END_IF;

		40:	(* cooler 2 stage 4 *)
			M_GK2V4			:=	1;
			M_GK2V5			:=	0;
			(* ON 5.stage *)
			IF	GK2_PLUS AND xR_TRIG_PLUS2.Q AND ST2_5	THEN
				schritt2	:=	50;
			END_IF;
			(* OFF 4.stage *)
			IF	GK2_MINUS AND (xR_TRIG_MINUS2.Q OR NOT ST2_5) THEN
				schritt2	:=	30;
			END_IF;

		50:	(* cooler 2 stage 5 *)
			M_GK2V5			:=	1;
			M_GK2V6			:=	0;
			(* ON 6.stage *)
			IF	GK2_PLUS AND xR_TRIG_PLUS2.Q AND ST2_6	THEN
				schritt2	:=	60;
			END_IF;
			(* OFF 5.stage *)
			IF	GK2_MINUS AND (xR_TRIG_MINUS2.Q OR NOT ST2_6) THEN
				schritt2	:=	40;
			END_IF;

		60:	(* cooler 2 stage 6 *)
			M_GK2V6			:=	1;
			M_GK2V7			:=	0;
			(* ON 7.stage *)
			IF	GK2_PLUS AND xR_TRIG_PLUS2.Q AND ST2_7	THEN
				schritt2	:=	70;
			END_IF;
			(* OFF 6.stage *)
			IF	GK2_MINUS AND (xR_TRIG_MINUS2.Q OR NOT ST2_7) THEN
				schritt2	:=	50;
			END_IF;

		70:	(* cooler 2 stage 7 *)
			M_GK2V7			:=	1;
			M_GK2V8			:=	0;
			(* ON 8.stage *)
			IF	GK2_PLUS AND xR_TRIG_PLUS2.Q AND ST2_8	THEN
				schritt2	:=	80;
			END_IF;
			(* OFF 7.stage *)
			IF	GK2_MINUS AND (xR_TRIG_MINUS2.Q OR NOT ST2_8) THEN
				schritt2	:=	60;
			END_IF;

		80:	(* cooler 2 stage 8 *)
			M_GK2V8			:=	1;
			M_GK2V9			:=	0;
			(* ON 9.stage *)
			IF	GK2_PLUS AND xR_TRIG_PLUS2.Q AND ST2_9	THEN
				schritt2	:=	90;
			END_IF;
			(* OFF 8.stage *)
			IF	GK2_MINUS AND (xR_TRIG_MINUS2.Q OR NOT ST2_9) THEN
				schritt2	:=	70;
			END_IF;

		90:	(* cooler 2 stage 9 *)
			M_GK2V9			:=	1;
			M_GK2V10		:=	0;
			(* ON 10.stage *)
			IF	GK2_PLUS AND xR_TRIG_PLUS2.Q AND ST2_10 THEN
				schritt2	:=	100;
			END_IF;
			(* OFF 9.stage *)
			IF	GK2_MINUS AND (xR_TRIG_MINUS2.Q OR NOT ST2_10)	THEN
				schritt2	:=	80;
			END_IF;

		100:(* cooler 2 stage 10 *)
			M_GK2V10		:=	1;
			M_GK2V11		:=	0;
			(* ON 11.stage *)
			IF	GK2_PLUS AND xR_TRIG_PLUS2.Q AND ST2_11 THEN
				schritt2	:=	110;
			END_IF;
			(* OFF 10.stage *)
			IF	GK2_MINUS AND (xR_TRIG_MINUS2.Q OR NOT ST2_11)	THEN
				schritt2	:=	90;
			END_IF;

		110:(* cooler 2 stage 11 *)
			M_GK2V11		:=	1;
			M_GK2V12		:=	0;
			(* ON 12.stage *)
			IF	GK2_PLUS AND xR_TRIG_PLUS2.Q AND ST2_12 THEN
				schritt2	:=	120;
			END_IF;
			(* OFF 11.stage *)
			IF	GK2_MINUS AND (xR_TRIG_MINUS2.Q OR NOT ST2_12)	THEN
				schritt2	:=	100;
			END_IF;

		120:(* cooler 2 stage 12 *)
			M_GK2V12		:=	1;
			M_GK2V13		:=	0;
			(* ON 13.stage *)
			IF	GK2_PLUS AND xR_TRIG_PLUS2.Q AND ST2_13 THEN
				schritt2	:=	130;
			END_IF;
			(* OFF 12.stage *)
			IF	GK2_MINUS AND (xR_TRIG_MINUS2.Q OR NOT ST2_13)	THEN
				schritt2	:=	110;
			END_IF;

		130:(* cooler 2 stage 13 *)
			M_GK2V13		:=	1;
			M_GK2V14		:=	0;
			(* ON 14.stage *)
			IF	GK2_PLUS AND xR_TRIG_PLUS2.Q AND ST2_14 THEN
				schritt2	:=	140;
			END_IF;
			(* OFF 13.stage *)
			IF	GK2_MINUS AND (xR_TRIG_MINUS2.Q OR NOT ST2_14)	THEN
				schritt2	:=	120;
			END_IF;

		140:(* cooler 2 stage 14 *)
			M_GK2V14		:=	1;
			M_GK2V15		:=	0;
			(* ON 15.stage *)
			IF	GK2_PLUS AND xR_TRIG_PLUS2.Q AND ST2_15 THEN
				schritt2	:=	150;
			END_IF;
			(* OFF 14.stage *)
			IF	GK2_MINUS AND (xR_TRIG_MINUS2.Q OR NOT ST2_15)	THEN
				schritt2	:=	130;
			END_IF;

		150:(* cooler 2 stage 15 *)
			M_GK2V15		:=	1;
			M_GK2V16		:=	0;
			(* ON 16.stage *)
			IF	GK2_PLUS AND xR_TRIG_PLUS2.Q AND ST2_16 THEN
				schritt2	:=	160;
			END_IF;
			(* OFF 15.stage *)
			IF	GK2_MINUS AND (xR_TRIG_MINUS2.Q OR NOT ST2_16)	THEN
				schritt2	:=	140;
			END_IF;

		160:(* cooler 2 stage 16 *)
			M_GK2V16		:=	1;
			(* OFF 16.stage *)
			IF	GK2_MINUS THEN
				schritt2	:=	150;
			END_IF;
		END_CASE;

		(* charge cooler 2 pump
		GK2P_EIN			:=	M_GK2V1; *)

		(* connection cooler stages to sequencing - charge cooler 2 *)
		GK2_ST1		:=	M_GK2V1;

		GK2_ST2		:=	M_GK2V1 AND gk2_anfhbt[2] OR
						M_GK2V2;

		GK2_ST3		:=	M_GK2V1 AND gk2_anfhbt[3] OR
						M_GK2V2 AND gk2_anfhbt[2] OR
						M_GK2V3;

		GK2_ST4		:=	M_GK2V1 AND gk2_anfhbt[4] OR
						M_GK2V2 AND gk2_anfhbt[3] OR
						M_GK2V3 AND gk2_anfhbt[2] OR
						M_GK2V4;

		GK2_ST5		:=	M_GK2V1 AND gk2_anfhbt[5] OR
						M_GK2V2 AND gk2_anfhbt[4] OR
						M_GK2V3 AND gk2_anfhbt[3] OR
						M_GK2V4 AND gk2_anfhbt[2] OR
						M_GK2V5;

		GK2_ST6		:=	M_GK2V1 AND gk2_anfhbt[6] OR
						M_GK2V2 AND gk2_anfhbt[5] OR
						M_GK2V3 AND gk2_anfhbt[4] OR
						M_GK2V4 AND gk2_anfhbt[3] OR
						M_GK2V5 AND gk2_anfhbt[2] OR
						M_GK2V6;

		GK2_ST7		:=	M_GK2V1 AND gk2_anfhbt[7] OR
						M_GK2V2 AND gk2_anfhbt[6] OR
						M_GK2V3 AND gk2_anfhbt[5] OR
						M_GK2V4 AND gk2_anfhbt[4] OR
						M_GK2V5 AND gk2_anfhbt[3] OR
						M_GK2V6 AND gk2_anfhbt[2] OR
						M_GK2V7;

		GK2_ST8		:=	M_GK2V1 AND gk2_anfhbt[8] OR
						M_GK2V2 AND gk2_anfhbt[7] OR
						M_GK2V3 AND gk2_anfhbt[6] OR
						M_GK2V4 AND gk2_anfhbt[5] OR
						M_GK2V5 AND gk2_anfhbt[4] OR
						M_GK2V6 AND gk2_anfhbt[3] OR
						M_GK2V7 AND gk2_anfhbt[2] OR
						M_GK2V8;

		GK2_ST9		:=	M_GK2V1 AND gk2_anfhbt[9] OR
						M_GK2V2 AND gk2_anfhbt[8] OR
						M_GK2V3 AND gk2_anfhbt[7] OR
						M_GK2V4 AND gk2_anfhbt[6] OR
						M_GK2V5 AND gk2_anfhbt[5] OR
						M_GK2V6 AND gk2_anfhbt[4] OR
						M_GK2V7 AND gk2_anfhbt[3] OR
						M_GK2V8 AND gk2_anfhbt[2] OR
						M_GK2V9;

		GK2_ST10	:=	M_GK2V1 AND gk2_anfhbt[10] OR
						M_GK2V2 AND gk2_anfhbt[9]  OR
						M_GK2V3 AND gk2_anfhbt[8]  OR
						M_GK2V4 AND gk2_anfhbt[7]  OR
						M_GK2V5 AND gk2_anfhbt[6]  OR
						M_GK2V6 AND gk2_anfhbt[5]  OR
						M_GK2V7 AND gk2_anfhbt[4]  OR
						M_GK2V8 AND gk2_anfhbt[3]  OR
						M_GK2V9 AND gk2_anfhbt[2]  OR
						M_GK2V10;

		GK2_ST11	:=	M_GK2V1  AND gk2_anfhbt[11] OR
						M_GK2V2  AND gk2_anfhbt[10] OR
						M_GK2V3  AND gk2_anfhbt[9]  OR
						M_GK2V4  AND gk2_anfhbt[8]  OR
						M_GK2V5  AND gk2_anfhbt[7]  OR
						M_GK2V6  AND gk2_anfhbt[6]  OR
						M_GK2V7  AND gk2_anfhbt[5]  OR
						M_GK2V8  AND gk2_anfhbt[4]  OR
						M_GK2V9  AND gk2_anfhbt[3]  OR
						M_GK2V10 AND gk2_anfhbt[2]  OR
						M_GK2V11;

		GK2_ST12	:=	M_GK2V1  AND gk2_anfhbt[12] OR
						M_GK2V2  AND gk2_anfhbt[11] OR
						M_GK2V3  AND gk2_anfhbt[10] OR
						M_GK2V4  AND gk2_anfhbt[9]  OR
						M_GK2V5  AND gk2_anfhbt[8]  OR
						M_GK2V6  AND gk2_anfhbt[7]  OR
						M_GK2V7  AND gk2_anfhbt[6]  OR
						M_GK2V8  AND gk2_anfhbt[5]  OR
						M_GK2V9  AND gk2_anfhbt[4]  OR
						M_GK2V10 AND gk2_anfhbt[3]  OR
						M_GK2V11 AND gk2_anfhbt[2]  OR
						M_GK2V12;

		GK2_ST13	:=	M_GK2V1  AND gk2_anfhbt[13] OR
						M_GK2V2  AND gk2_anfhbt[12] OR
						M_GK2V3  AND gk2_anfhbt[11] OR
						M_GK2V4  AND gk2_anfhbt[10] OR
						M_GK2V5  AND gk2_anfhbt[9]  OR
						M_GK2V6  AND gk2_anfhbt[8]  OR
						M_GK2V7  AND gk2_anfhbt[7]  OR
						M_GK2V8  AND gk2_anfhbt[6]  OR
						M_GK2V9  AND gk2_anfhbt[5]  OR
						M_GK2V10 AND gk2_anfhbt[4]  OR
						M_GK2V11 AND gk2_anfhbt[3]  OR
						M_GK2V12 AND gk2_anfhbt[2]  OR
						M_GK2V13;

		GK2_ST14	:=	M_GK2V1  AND gk2_anfhbt[14] OR
						M_GK2V2  AND gk2_anfhbt[13] OR
						M_GK2V3  AND gk2_anfhbt[12] OR
						M_GK2V4  AND gk2_anfhbt[11] OR
						M_GK2V5  AND gk2_anfhbt[10] OR
						M_GK2V6  AND gk2_anfhbt[9]  OR
						M_GK2V7  AND gk2_anfhbt[8]  OR
						M_GK2V8  AND gk2_anfhbt[7]  OR
						M_GK2V9  AND gk2_anfhbt[6]  OR
						M_GK2V10 AND gk2_anfhbt[5]  OR
						M_GK2V11 AND gk2_anfhbt[4]  OR
						M_GK2V12 AND gk2_anfhbt[3]  OR
						M_GK2V13 AND gk2_anfhbt[2]  OR
						M_GK2V14;

		GK2_ST15	:=	M_GK2V1  AND gk2_anfhbt[15] OR
						M_GK2V2  AND gk2_anfhbt[14] OR
						M_GK2V3  AND gk2_anfhbt[13] OR
						M_GK2V4  AND gk2_anfhbt[12] OR
						M_GK2V5  AND gk2_anfhbt[11] OR
						M_GK2V6  AND gk2_anfhbt[10] OR
						M_GK2V7  AND gk2_anfhbt[9]  OR
						M_GK2V8  AND gk2_anfhbt[8]  OR
						M_GK2V9  AND gk2_anfhbt[7]  OR
						M_GK2V10 AND gk2_anfhbt[6]  OR
						M_GK2V11 AND gk2_anfhbt[5]  OR
						M_GK2V12 AND gk2_anfhbt[4]  OR
						M_GK2V13 AND gk2_anfhbt[3]  OR
						M_GK2V14 AND gk2_anfhbt[2]  OR
						M_GK2V15;

		GK2_ST16	:=	M_GK2V1  AND gk2_anfhbt[16] OR
						M_GK2V2  AND gk2_anfhbt[15] OR
						M_GK2V3  AND gk2_anfhbt[14] OR
						M_GK2V4  AND gk2_anfhbt[13] OR
						M_GK2V5  AND gk2_anfhbt[12] OR
						M_GK2V6  AND gk2_anfhbt[11] OR
						M_GK2V7  AND gk2_anfhbt[10] OR
						M_GK2V8  AND gk2_anfhbt[9]  OR
						M_GK2V9  AND gk2_anfhbt[8]  OR
						M_GK2V10 AND gk2_anfhbt[7]  OR
						M_GK2V11 AND gk2_anfhbt[6]  OR
						M_GK2V12 AND gk2_anfhbt[5]  OR
						M_GK2V13 AND gk2_anfhbt[4]  OR
						M_GK2V14 AND gk2_anfhbt[3]  OR
						M_GK2V15 AND gk2_anfhbt[2]  OR
						M_GK2V16;

		(* copy for summation - charge cooler 2 *)
		GK2ST[1]	:=	BOOL_TO_USINT(M_GK2V1);
		GK2ST[2]	:=	BOOL_TO_USINT(M_GK2V2);
		GK2ST[3]	:=	BOOL_TO_USINT(M_GK2V3);
		GK2ST[4]	:=	BOOL_TO_USINT(M_GK2V4);
		GK2ST[5]	:=	BOOL_TO_USINT(M_GK2V5);
		GK2ST[6]	:=	BOOL_TO_USINT(M_GK2V6);
		GK2ST[7]	:=	BOOL_TO_USINT(M_GK2V7);
		GK2ST[8]	:=	BOOL_TO_USINT(M_GK2V8);
		GK2ST[9]	:=	BOOL_TO_USINT(M_GK2V9);
		GK2ST[10]	:=	BOOL_TO_USINT(M_GK2V10);
		GK2ST[11]	:=	BOOL_TO_USINT(M_GK2V11);
		GK2ST[12]	:=	BOOL_TO_USINT(M_GK2V12);
		GK2ST[13]	:=	BOOL_TO_USINT(M_GK2V13);
		GK2ST[14]	:=	BOOL_TO_USINT(M_GK2V14);
		GK2ST[15]	:=	BOOL_TO_USINT(M_GK2V15);
		GK2ST[16]	:=	BOOL_TO_USINT(M_GK2V16);

		(* ON/OFF coolerstage *)
		summe2 := 0;
		FOR i:=	1 TO 16 BY 1 DO
			summe2 := summe2 + GK2ST[i];
		END_FOR;

		plus2 :=	0;
		IF summe2 > summe2_old THEN
			plus2 := 1;
		END_IF;

		minus2 := 0;
		IF summe2 < summe2_old THEN
			minus2 := 1;
		END_IF;

		summe2_old := summe2;

	END_IF;

	(*----------------------------------------------------------------------------*)
	(* BEL Standard *)
	(* demand heating charge cooler ventilation  *)
	OUT_HC.tChC_Heating.Do := ((NOT bT_AirOutdoor_Hi1 AND Para.bT_AirOutdoor_Active)
								 OR IN_HC.tManAuxCtr.bChC_Heating)		(* Manual operating auxiliaries control - Handbedienebene *)
							AND	NOT IN_HC.bMsg1031
							AND NOT IN_HC.bMsg1053
							AND NOT IN_HC.bMsg1054;

	OUT_HC.tChC2_Heating.Do :=((NOT bT_AirOutdoor_Hi1 AND Para.bT_AirOutdoor_Active)
								 OR IN_HC.tManAuxCtr.bChC2_Heating)	(* Manual operating auxiliaries control - Handbedienebene *)
							AND	NOT IN_HC.bMsg1031
							AND NOT IN_HC.bMsg1053
							AND NOT IN_HC.bMsg1054;
	(*----------------------------------------------------------------------------*)

END_PROGRAM
```

#### ChC.var
```iecst
VAR
	rValvePos : REAL := 0.0; (*valve position*)
	GK_reg : USINT;
	minus : BOOL := 0;
	plus : BOOL := 0;
	REG_INVERT : BOOL;
	ST_10 : BOOL;
	ST_9 : BOOL;
	ST_8 : BOOL;
	ST_3 : BOOL;
	ST_4 : BOOL;
	ST_5 : BOOL;
	ST_7 : BOOL;
	ST_6 : BOOL;
	ST_2 : BOOL;
	ST_11 : BOOL;
	ST_16 : BOOL;
	ST_15 : BOOL;
	ST_1 : BOOL;
	Temp_KuehlerAustritt : BOOL;
	ST_12 : BOOL;
	ST_13 : BOOL;
	ST_14 : BOOL;
	gk_anfhbt : ARRAY[0..16] OF BOOL;
	xGRMax_Ventpos : GR_MAXR;
	xGRMax_Ventpos2 : GR_MAXR;
	xGRMin_Ventpos : GR_MINR;
	xR_TRIG_PLUS : R_TRIG;
	xR_TRIG_MINUS : R_TRIG;
	xTOF_MINUS : TOF;
	xTOF_GK_AUS : TOF;
	xTOF_PLUS : TOF;
	zw : UDINT;
	summe_old : USINT := 0;
	summe : USINT;
	F_SPSR : USINT;
	Anz_GK_vent : USINT;
	i : USINT;
	schritt : USINT := 0;
	Anz_GK_st : USINT;
	GKST : ARRAY[0..16] OF USINT;
	FA_INIT_2 : WDtoBIT;
	FA_INIT_3 : WDtoBIT;
	FA_INIT_1 : WDtoBIT;
	GK2_reg : USINT;
	gk2_anfhbt : ARRAY[0..16] OF BOOL;
	Anz_GK2_st : USINT;
	FA2_INIT_1 : WDtoBIT;
	FA2_INIT_2 : WDtoBIT;
	FA2_INIT_3 : WDtoBIT;
	ST2_1 : BOOL;
	ST2_2 : BOOL;
	ST2_3 : BOOL;
	ST2_4 : BOOL;
	ST2_5 : BOOL;
	ST2_6 : BOOL;
	ST2_7 : BOOL;
	ST2_8 : BOOL;
	ST2_9 : BOOL;
	ST2_10 : BOOL;
	ST2_11 : BOOL;
	ST2_12 : BOOL;
	ST2_13 : BOOL;
	ST2_14 : BOOL;
	ST2_15 : BOOL;
	ST2_16 : BOOL;
	Anz_GK2_vent : USINT;
	F2_SPSR : USINT;
	rValvePos2 : REAL := 0.0; (*valve position*)
	REG2_INVERT : BOOL;
	xGRMax2_Ventpos : GR_MAXR;
	xTOF_GK2_AUS : TOF;
	xGRMax2_Ventpos2 : GR_MAXR;
	xGRMin2_Ventpos : GR_MINR;
	xTOF_PLUS2 : TOF;
	xTOF_MINUS2 : TOF;
	plus2 : BOOL := 0;
	minus2 : BOOL := 0;
	xR_TRIG_PLUS2 : R_TRIG;
	xR_TRIG_MINUS2 : R_TRIG;
	schritt2 : USINT := 0;
	GK2ST : ARRAY[0..16] OF USINT;
	summe2_old : USINT := 0;
	summe2 : USINT;
END_VAR
```

### Program Logical/HeatingCooling/ChC_Seq (IEC, version 4.07.0) - charge cooler sequence

#### ChC_SeqCyclic.st
```iecst
(*******************************************************************************
ChC_Seq			charge cooler sequence for 16 stages

This code is confidential AND proprietary to the INNIO Company.
It may NOT be used in any form, OR reproduced in any manner,
without written permission of the INNIO Company.
Copyright, INNIO Company, 2019

Customized modifications: -
------------------------

History:
-------
V0.1 	31-01-2003	Thaler, generated
     	21-03-2003	Thaler, last modification
V1.82	06-10-2003	LH, bits für Anzeige auf VISU,
						Variable für XT-Anzeige
V2.071a	31-03-2005	LH, Variable für Freigabe XT-Anzeige
V2.30	24-01-2008	LH, Variable für Freigabe XT-Anzeige gelöscht (Parameter!)
V3.99.0	21.02.2013	lettenb.	gkv_seq -> ChC_Seq renamed
V4.03.0 07.08.2015  Denk		Manual operating auxiliaries control functionality added
V4.07.0	09.08.2018	Schmid		2nd low temperature charge cooling circuit added

Instructions for use:
--------------------

Outstandings:
------------
*******************************************************************************)

PROGRAM _CYCLIC

	GK_Var := INT_TO_USINT(LIMIT(0, Para.iChC_OpMode, 2));
	GK2_Var := INT_TO_USINT(LIMIT(0, Para.iChC2_OpMode, 22));

	(* Manual operating auxiliaries control - Handbedienebene *)
	FOR i:= 1 TO Para.iChC_NumStages BY 1 DO
		IF 	(GK_Var < 3) THEN
			GK_ST1_ManAuxCtr:=  IN_HC.tManAuxCtr.bChC_DemFan;
			GK_ST2_ManAuxCtr:=  IN_HC.tManAuxCtr.bChC_DemFan;
			GK_ST3_ManAuxCtr:=  IN_HC.tManAuxCtr.bChC_DemFan;
			GK_ST4_ManAuxCtr:=  IN_HC.tManAuxCtr.bChC_DemFan;
			GK_ST5_ManAuxCtr:=  IN_HC.tManAuxCtr.bChC_DemFan;
			GK_ST6_ManAuxCtr:=  IN_HC.tManAuxCtr.bChC_DemFan;
			GK_ST7_ManAuxCtr:=  IN_HC.tManAuxCtr.bChC_DemFan;
			GK_ST8_ManAuxCtr:=  IN_HC.tManAuxCtr.bChC_DemFan;
			GK_ST9_ManAuxCtr:=  IN_HC.tManAuxCtr.bChC_DemFan;
			GK_ST10_ManAuxCtr:= IN_HC.tManAuxCtr.bChC_DemFan;
			GK_ST11_ManAuxCtr:= IN_HC.tManAuxCtr.bChC_DemFan;
			GK_ST12_ManAuxCtr:= IN_HC.tManAuxCtr.bChC_DemFan;
			GK_ST13_ManAuxCtr:= IN_HC.tManAuxCtr.bChC_DemFan;
			GK_ST14_ManAuxCtr:= IN_HC.tManAuxCtr.bChC_DemFan;
			GK_ST15_ManAuxCtr:= IN_HC.tManAuxCtr.bChC_DemFan;
			GK_ST16_ManAuxCtr:= IN_HC.tManAuxCtr.bChC_DemFan;

			IF IN_HC.tManAuxCtr.bChC_DemFan = TRUE THEN
				iSumChC_Stages_ManAuxCtr := Para.iChC_NumStages;
			ELSE
				iSumChC_Stages_ManAuxCtr := 0;
			END_IF;
		END_IF;
	END_FOR;

	(* connection of in-/outputs *)
	EN[1]  := GK_ST_1;
	EN[2]  := GK_ST_2;
	EN[3]  := GK_ST_3;
	EN[4]  := GK_ST_4;
	EN[5]  := GK_ST_5;
	EN[6]  := GK_ST_6;
	EN[7]  := GK_ST_7;
	EN[8]  := GK_ST_8;
	EN[9]  := GK_ST_9;
	EN[10] := GK_ST_10;
	EN[11] := GK_ST_11;
	EN[12] := GK_ST_12;
	EN[13] := GK_ST_13;
	EN[14] := GK_ST_14;
	EN[15] := GK_ST_15;
	EN[16] := GK_ST_16;

	IN[1]  := GK_ST1;
	IN[2]  := GK_ST2;
	IN[3]  := GK_ST3;
	IN[4]  := GK_ST4;
	IN[5]  := GK_ST5;
	IN[6]  := GK_ST6;
	IN[7]  := GK_ST7;
	IN[8]  := GK_ST8;
	IN[9]  := GK_ST9;
	IN[10] := GK_ST10;
	IN[11] := GK_ST11;
	IN[12] := GK_ST12;
	IN[13] := GK_ST13;
	IN[14] := GK_ST14;
	IN[15] := GK_ST15;
	IN[16] := GK_ST16;

	(* Para.iChC2_OpMode = 11, 12:	combi cooler for LT cooling water circuits
	   -> activate cooler stage IF request from one OF the circuits
	   -> deactivate cooler stage only IF request from both circuits *)
	IF Para.bAuxChC2_Visible AND GK2_Var/10 = 1 THEN
		IN[1]  := IN[1] OR GK2_ST1;
		IN[2]  := IN[2] OR GK2_ST2;
		IN[3]  := IN[3] OR GK2_ST3;
		IN[4]  := IN[4] OR GK2_ST4;
		IN[5]  := IN[5] OR GK2_ST5;
		IN[6]  := IN[6] OR GK2_ST6;
		IN[7]  := IN[7] OR GK2_ST7;
		IN[8]  := IN[8] OR GK2_ST8;
		IN[9]  := IN[9] OR GK2_ST9;
		IN[10] := IN[10] OR GK2_ST10;
		IN[11] := IN[11] OR GK2_ST11;
		IN[12] := IN[12] OR GK2_ST12;
		IN[13] := IN[13] OR GK2_ST13;
		IN[14] := IN[14] OR GK2_ST14;
		IN[15] := IN[15] OR GK2_ST15;
		IN[16] := IN[16] OR GK2_ST16;
	END_IF;

	OUT_HC.tChC_DemFan1.Do := Q[1] OR GK_ST1_ManAuxCtr;
	OUT_HC.tChC_DemFan2.Do := Q[2] OR GK_ST2_ManAuxCtr;
	OUT_HC.tChC_DemFan3.Do := Q[3] OR GK_ST3_ManAuxCtr;
	OUT_HC.tChC_DemFan4.Do := Q[4] OR GK_ST4_ManAuxCtr;
	OUT_HC.tChC_DemFan5.Do := Q[5] OR GK_ST5_ManAuxCtr;
	OUT_HC.tChC_DemFan6.Do := Q[6] OR GK_ST6_ManAuxCtr;
	OUT_HC.tChC_DemFan7.Do := Q[7] OR GK_ST7_ManAuxCtr;
	OUT_HC.tChC_DemFan8.Do := Q[8] OR GK_ST8_ManAuxCtr;
	OUT_HC.tChC_DemFan9.Do := Q[9] OR GK_ST9_ManAuxCtr;
	OUT_HC.tChC_DemFan10.Do := Q[10] OR GK_ST10_ManAuxCtr;
	OUT_HC.tChC_DemFan11.Do := Q[11] OR GK_ST11_ManAuxCtr;
	OUT_HC.tChC_DemFan12.Do := Q[12] OR GK_ST12_ManAuxCtr;
	OUT_HC.tChC_DemFan13.Do := Q[13] OR GK_ST13_ManAuxCtr;
	OUT_HC.tChC_DemFan14.Do := Q[14] OR GK_ST14_ManAuxCtr;
	OUT_HC.tChC_DemFan15.Do := Q[15] OR GK_ST15_ManAuxCtr;
	OUT_HC.tChC_DemFan16.Do := Q[16] OR GK_ST16_ManAuxCtr;

	(******************************************************************************)

	and_16b (ADR(EN), ADR(Q), ADR(Q));		(* switch off "Q" if "EN" is FALSE:   "Q" := "EN" AND "Q" *)
	andnt_16b (ADR(EN), ADR(Q), ADR(RDY));	(* enabled outputs with status FALSE: "RDY" := "EN" AND NOT "Q" *)

	(* SEQU_C = stage number for stage numbers > iPriorityStage *)
	FOR i := (iPriorityStage + 1) TO 16 BY 1 DO
		SEQU_C[i] := i;
	END_FOR;

	(* SEQU_C = stage number + 100 for stage numbers <= iPriorityStage *)
	FOR i := iPriorityStage TO 1 BY -1 DO
		 SEQU_C[i] := i + 100;
	END_FOR;

	min_16di (ADR(RDY), ADR(SEQU_C), ADR(NEXT_ON));	(* stage for next on  as BOOL *)
	min_16di (ADR(Q), ADR(SEQU_C), ADR(NEXT_OFF)); 	(* stage for next off as BOOL *)

	iNextOn   := max_i_16b (ADR(NEXT_ON)); 			(* stage for next on  as INT  *)
	iNextOff  := max_i_16b (ADR(NEXT_OFF));			(* stage for next off as INT  *)

	iIN := max_i_16b (ADR(IN));						(* input : number of stages as INT *)
	iQ  := sum_16b (ADR(Q));   						(* output: number of stages as INT *)

	IF (iIN > iQ) THEN
		Q[iNextOn] := TRUE;
		iPriorityStage := iNextOn;
	END_IF;

	IF (iIN < iQ) THEN
		Q[iNextOff] := FALSE;
	END_IF;

	(******************************************************************************)

	(* bits für Anzeige auf VISU *)

	summe := 0;
	FOR i:= 1 TO 16 BY 1 DO
		summe := summe + Q[i];
	END_FOR;

	GK_byte1 := FALSE;
	GK_byte2 := FALSE;

	GK_bit10 := FALSE;
	GK_bit11 := FALSE;
	GK_bit12 := FALSE;

	GK_bit20 := FALSE;
	GK_bit21 := FALSE;
	GK_bit22 := FALSE;

	IF	(summe > 0) AND (summe < 9) THEN
		GK_byte1 := TRUE;
	END_IF;

	IF	((summe = 2) OR (summe = 4) OR (summe = 6) OR (summe = 8)) THEN
		GK_bit10 := TRUE;
	END_IF;

	IF	((summe = 3) OR (summe = 4) OR (summe = 7) OR (summe = 8)) THEN
		GK_bit11 := TRUE;
	END_IF;

	IF	((summe = 5) OR (summe = 6) OR (summe = 7) OR (summe = 8)) THEN
		GK_bit12 := TRUE;
	END_IF;

	IF	(summe > 8) THEN
		GK_byte2 := TRUE;
	END_IF;

	IF	((summe = 10) OR (summe = 12) OR (summe = 14) OR (summe = 16)) THEN
		GK_bit20 := TRUE;
	END_IF;

	IF	((summe = 11) OR (summe = 12) OR (summe = 15) OR (summe = 16)) THEN
		GK_bit21 := TRUE;
	END_IF;

	IF	((summe = 13) OR (summe = 14) OR (summe = 15) OR (summe = 16)) THEN
		GK_bit22 := TRUE;
	END_IF;

	IF iSumChC_Stages_ManAuxCtr > 0 THEN
		iSumChC_Stages := iSumChC_Stages_ManAuxCtr; 	(* Manual operating auxiliaries control - Handbedienebene to vis *)
	ELSE
		iSumChC_Stages := summe;						(* to vis *)
	END_IF;

	(******************************************************************************)
	(* charge cooler 2 stage sequence control
	   Para.iChC2_OpMode = 21, 22:	2 separate LT charge cooling water circuits, 2 coolers
									-> independent cooler stage control *)
	IF GK2_Var > 20 AND Para.bAuxChC2_Visible THEN
		(* Manual operating auxiliaries control - Handbedienebene *)
		GK2_ST1_ManAuxCtr	:=  IN_HC.tManAuxCtr.bChC2_DemFan;
		GK2_ST2_ManAuxCtr	:=  IN_HC.tManAuxCtr.bChC2_DemFan;
		GK2_ST3_ManAuxCtr	:=  IN_HC.tManAuxCtr.bChC2_DemFan;
		GK2_ST4_ManAuxCtr	:=  IN_HC.tManAuxCtr.bChC2_DemFan;
		GK2_ST5_ManAuxCtr	:=  IN_HC.tManAuxCtr.bChC2_DemFan;
		GK2_ST6_ManAuxCtr	:=  IN_HC.tManAuxCtr.bChC2_DemFan;
		GK2_ST7_ManAuxCtr	:=  IN_HC.tManAuxCtr.bChC2_DemFan;
		GK2_ST8_ManAuxCtr	:=  IN_HC.tManAuxCtr.bChC2_DemFan;
		GK2_ST9_ManAuxCtr	:=  IN_HC.tManAuxCtr.bChC2_DemFan;
		GK2_ST10_ManAuxCtr	:=	IN_HC.tManAuxCtr.bChC2_DemFan;
		GK2_ST11_ManAuxCtr	:=	IN_HC.tManAuxCtr.bChC2_DemFan;
		GK2_ST12_ManAuxCtr	:=	IN_HC.tManAuxCtr.bChC2_DemFan;
		GK2_ST13_ManAuxCtr	:=	IN_HC.tManAuxCtr.bChC2_DemFan;
		GK2_ST14_ManAuxCtr	:=	IN_HC.tManAuxCtr.bChC2_DemFan;
		GK2_ST15_ManAuxCtr	:=	IN_HC.tManAuxCtr.bChC2_DemFan;
		GK2_ST16_ManAuxCtr	:=	IN_HC.tManAuxCtr.bChC2_DemFan;

		IF IN_HC.tManAuxCtr.bChC2_DemFan THEN
			iSumChC2_Stages_ManAuxCtr := Para.iChC2_NumStages;
		ELSE
			iSumChC2_Stages_ManAuxCtr := 0;
		END_IF;

		(* connection of in-/outputs *)
		EN2[1]  := GK2_ST_1;
		EN2[2]  := GK2_ST_2;
		EN2[3]  := GK2_ST_3;
		EN2[4]  := GK2_ST_4;
		EN2[5]  := GK2_ST_5;
		EN2[6]  := GK2_ST_6;
		EN2[7]  := GK2_ST_7;
		EN2[8]  := GK2_ST_8;
		EN2[9]  := GK2_ST_9;
		EN2[10] := GK2_ST_10;
		EN2[11] := GK2_ST_11;
		EN2[12] := GK2_ST_12;
		EN2[13] := GK2_ST_13;
		EN2[14] := GK2_ST_14;
		EN2[15] := GK2_ST_15;
		EN2[16] := GK2_ST_16;

		IN2[1]  := GK2_ST1;
		IN2[2]  := GK2_ST2;
		IN2[3]  := GK2_ST3;
		IN2[4]  := GK2_ST4;
		IN2[5]  := GK2_ST5;
		IN2[6]  := GK2_ST6;
		IN2[7]  := GK2_ST7;
		IN2[8]  := GK2_ST8;
		IN2[9]  := GK2_ST9;
		IN2[10] := GK2_ST10;
		IN2[11] := GK2_ST11;
		IN2[12] := GK2_ST12;
		IN2[13] := GK2_ST13;
		IN2[14] := GK2_ST14;
		IN2[15] := GK2_ST15;
		IN2[16] := GK2_ST16;

		OUT_HC.tChC2_DemFan1.Do		:= Q2[1]	OR GK2_ST1_ManAuxCtr;
		OUT_HC.tChC2_DemFan2.Do 	:= Q2[2]	OR GK2_ST2_ManAuxCtr;
		OUT_HC.tChC2_DemFan3.Do 	:= Q2[3]	OR GK2_ST3_ManAuxCtr;
		OUT_HC.tChC2_DemFan4.Do 	:= Q2[4]	OR GK2_ST4_ManAuxCtr;
		OUT_HC.tChC2_DemFan5.Do 	:= Q2[5]	OR GK2_ST5_ManAuxCtr;
		OUT_HC.tChC2_DemFan6.Do 	:= Q2[6]	OR GK2_ST6_ManAuxCtr;
		OUT_HC.tChC2_DemFan7.Do 	:= Q2[7]	OR GK2_ST7_ManAuxCtr;
		OUT_HC.tChC2_DemFan8.Do 	:= Q2[8]	OR GK2_ST8_ManAuxCtr;
		OUT_HC.tChC2_DemFan9.Do 	:= Q2[9]	OR GK2_ST9_ManAuxCtr;
		OUT_HC.tChC2_DemFan10.Do	:= Q2[10]	OR GK2_ST10_ManAuxCtr;
		OUT_HC.tChC2_DemFan11.Do 	:= Q2[11]	OR GK2_ST11_ManAuxCtr;
		OUT_HC.tChC2_DemFan12.Do 	:= Q2[12]	OR GK2_ST12_ManAuxCtr;
		OUT_HC.tChC2_DemFan13.Do	:= Q2[13]	OR GK2_ST13_ManAuxCtr;
		OUT_HC.tChC2_DemFan14.Do	:= Q2[14]	OR GK2_ST14_ManAuxCtr;
		OUT_HC.tChC2_DemFan15.Do	:= Q2[15]	OR GK2_ST15_ManAuxCtr;
		OUT_HC.tChC2_DemFan16.Do	:= Q2[16]	OR GK2_ST16_ManAuxCtr;

		(******************************************************************************)

		and_16b (ADR(EN2), ADR(Q2), ADR(Q2));		(* switch off "Q2" if "EN2" is FALSE:   "Q2" := "EN2" AND "Q2" *)
		andnt_16b (ADR(EN2), ADR(Q2), ADR(RDY2));	(* enabled outputs with status FALSE: "RDY2" := "EN2" AND NOT "Q2" *)

		(* SEQU_C2 = stage number for stage numbers > iPriorityStage2 *)
		FOR i := (iPriorityStage2 + 1) TO 16 BY 1 DO
			SEQU_C2[i] := i;
		END_FOR;

		(* SEQU_C2 = stage number + 100 for stage numbers <= iPriorityStage2 *)
		FOR i := iPriorityStage2 TO 1 BY -1 DO
			 SEQU_C2[i] := i + 100;
		END_FOR;

		min_16di (ADR(RDY2), ADR(SEQU_C2), ADR(NEXT_ON2));	(* stage for next on  as BOOL *)
		min_16di (ADR(Q2), ADR(SEQU_C2), ADR(NEXT_OFF2)); 	(* stage for next off as BOOL *)

		iNextOn2   := max_i_16b (ADR(NEXT_ON2)); 			(* stage for next on  as INT  *)
		iNextOff2  := max_i_16b (ADR(NEXT_OFF2));			(* stage for next off as INT  *)

		iIN2 := max_i_16b (ADR(IN2));						(* input : number of stages as INT *)
		iQ2  := sum_16b (ADR(Q2));   						(* output: number of stages as INT *)

		IF (iIN2 > iQ2) THEN
			Q2[iNextOn2] := TRUE;
			iPriorityStage2 := iNextOn2;
		END_IF;

		IF (iIN2 < iQ2) THEN
			Q2[iNextOff2] := FALSE;
		END_IF;

		(******************************************************************************)

		(* Anzeige auf VISU *)

		summe2 := 0;
		FOR i:= 1 TO 16 BY 1 DO
			summe2 := summe2 + Q2[i];
		END_FOR;

		IF iSumChC2_Stages_ManAuxCtr > 0 THEN
			iSumChC2_Stages := iSumChC2_Stages_ManAuxCtr; 	(* Manual operating auxiliaries control - Handbedienebene to vis *)
		ELSE
			iSumChC2_Stages := summe2;						(* to vis *)
		END_IF;
	END_IF;

END_PROGRAM
```

#### ChC_Seq.var
```iecst
VAR
	GK_bit10 : BOOL := 0; (* Anzeige-Bit *)
	GK_bit11 : BOOL := 0; (* Anzeige-Bit *)
	GK_bit12 : BOOL := 0; (* Anzeige-Bit *)
	GK_bit20 : BOOL := 0; (* Anzeige-Bit *)
	GK_bit21 : BOOL := 0; (* Anzeige-Bit *)
	GK_bit22 : BOOL := 0; (* Anzeige-Bit *)
	GK_byte1 : BOOL := 0; (* Anzeige-Byte *)
	GK_byte2 : BOOL := 0; (* Anzeige-Byte *)
	IN : ARRAY[0..16] OF BOOL;
	Q : ARRAY[0..16] OF BOOL;
	RDY : ARRAY[0..16] OF BOOL;
	EN : ARRAY[0..16] OF BOOL;
	iQ : INT;
	iIN : INT;
	iPriorityStage : INT;
	SEQU_C : ARRAY[0..16] OF DINT;
	NEXT_ON : ARRAY[0..16] OF BOOL;
	NEXT_OFF : ARRAY[0..16] OF BOOL;
	i : INT;
	iNextOn : INT;
	iNextOff : INT;
	summe : USINT := 0;
	GK_Var : USINT; (* charge cooler variation *)
	iSumChC_Stages_ManAuxCtr : INT; (*summary charge cooler stages from Manual operating auxiliaries control *)
	iSumChC2_Stages_ManAuxCtr : INT; (*summary charge cooler 2 stages from Manual operating auxiliaries control *)
	EN2 : ARRAY[0..16] OF BOOL;
	IN2 : ARRAY[0..16] OF BOOL;
	Q2 : ARRAY[0..16] OF BOOL;
	RDY2 : ARRAY[0..16] OF BOOL;
	iPriorityStage2 : INT;
	SEQU_C2 : ARRAY[0..16] OF DINT;
	iNextOn2 : INT;
	iNextOff2 : INT;
	NEXT_ON2 : ARRAY[0..16] OF BOOL;
	NEXT_OFF2 : ARRAY[0..16] OF BOOL;
	iQ2 : INT;
	iIN2 : INT;
	summe2 : USINT := 0;
	GK2_Var : USINT; (* charge cooler 2 variant *)
END_VAR
```

### Program Logical/HeatingCooling/Cnt_P_Heat (IEC, version 4.03.0) - counter heat power

#### Cnt_P_HeatCyclic.st
```iecst
(*******************************************************************************
Cnt_P_Heat		counter for heat power engine heat water circuit

This code is confidential AND proprietary to the INNIO Company.
It may NOT be used in any form, OR reproduced in any manner,
without written permission of the INNIO Company.
Copyright, INNIO Company, 2019

Customized modifications: -
------------------------

History:
-------
V4.03.0		Stary 		created
			lettenb.	xImp_Cnt_P_Heat: function call brackets missing, bugfix

Instructions for use:
--------------------

Outstandings:
------------
*******************************************************************************)

PROGRAM _CYCLIC

	(* counter heat power engine heat water circuit *)
	xImp_Cnt_P_Heat(CLK:= IN_HC.tP_Heat_Imp.Di);

	(* counter heat power engine heat water circuit *)
	IF xImp_Cnt_P_Heat.Q THEN
		(* increase counter *)
		MM2VIS.iCnt_P_Heat := MM2VIS.iCnt_P_Heat + REAL_TO_INT(Para.rImpVal_Cnt_P_Heat);
		(* check limits *)
		IF MM2VIS.iCnt_P_Heat >= 1000000000 THEN
			MM2VIS.iCnt_P_Heat := MM2VIS.iCnt_P_Heat - 1000000000;		(* check upper limit *)
		ELSIF MM2VIS.iCnt_P_Heat <= -1000000000 THEN
			MM2VIS.iCnt_P_Heat := MM2VIS.iCnt_P_Heat + 1000000000;		(* check lower limit *)
		END_IF;
	END_IF;
	OUT_HC.iCnt_P_Heat	:= MM2VIS.iCnt_P_Heat;		(* MM2VIS = read/write = ausnahme damit vis abwärtskompatibel bleibt!!*)

END_PROGRAM
```

#### Cnt_P_Heat.var
```iecst
VAR
	xImp_Cnt_P_Heat : R_TRIG; (* R_TRIG heat counter *)
END_VAR
```

### Program Logical/HeatingCooling/Ctr_CDSu (IEC, version 4.11.0) - controller condensor circuit supply temperature

#### Ctr_CDSuCyclic.st
```iecst
(*******************************************************************************
Ctr_CDSu		controller condensor circuit supply temperature

This code is confidential and proprietary to the INNIO Company.
It may not be used in any form, or reproduced in any manner,
without the express written permission of the INNIO Company.
Copyright, INNIO Company, 2022

Customized modifications: -
------------------------

History:
-------
V4.03.0		27.07.2015	Plattner	task creation
V4.11.0		28.01.2022	Perktold	included plant controller upgrade

Instructions for use:
--------------------

Outstandings:
------------
(*******************************************************************************)

PROGRAM _CYCLIC

	(* Parameter *)
	Para.tCtr_CDSu.W_set;
	Para.tCtr_CDSu.W_set2;
	Para.tCtr_CDSu.W_min;
	Para.tCtr_CDSu.W_max;
	Para.tCtr_CDSu.dW_up;
	Para.tCtr_CDSu.dW_down;
	Para.tCtr_CDSu.deadband;
	Para.tCtr_CDSu.Y_min;
	Para.tCtr_CDSu.Y_max;
	Para.tCtr_CDSu.dY_max;
	Para.tCtr_CDSu.Y_block;
	Para.tCtr_CDSu.invert;
	Para.tCtr_CDSu.Kp;
	Para.tCtr_CDSu.Tn;
	Para.tCtr_CDSu.Tv;
	Para.tCtr_CDSu.Kp_GainScheduling;
	Para.tCtr_CDSu.Tn_GainScheduling;
	Para.tCtr_CDSu.Tv_GainScheduling;
	Para.tCtr_CDSu.t_min_pulse_down;
	Para.tCtr_CDSu.t_min_pulse_up;
	Para.tCtr_CDSu.t_period_down;
	Para.tCtr_CDSu.t_period_up;

	(* Input variables *)
	tCtr_CDSu_In				:= VIS2MM.tCtr_CDSu_In;			(* from vis *)

	(* Input from module *)
	tCtr_CDSu_In.enable			:=	Para.bCtr_CDSu
								AND	IN_HC.tPB2MM.bParaSetupOk
								AND IN_HC.bEng_Aux_Dem_CDR
								AND IN_HC.tT_CD_Su.GoodQual;
	tCtr_CDSu_In.W_ext_Active	:= tCtr_CDSu_In.W_ext_Active;	(* from vis *)
	tCtr_CDSu_In.W_ext			:= 0.0;
	tCtr_CDSu_In.Y_set_Active	:= NOT IN_HC.tT_CD_Su.GoodQual;
	tCtr_CDSu_In.Y_set			:= 1.0;
	tCtr_CDSu_In.X				:= IN_HC.tT_CD_Su.Ai;
	tCtr_CDSu_In.A				:= 0;
	tCtr_CDSu_In.W_set2_Active	:= FALSE;	(*Input to define which internal setpoint will be used TRUE = use the 2nd set point | FALSE use the normal "1st" one*)
	tCtr_CDSu_In.GainScheduling	:= 0.0;		(*Input for Gain Scheduling: 0.0 = use 100% of the Standard PID-Parameters | 1.0 = use 100% of the GainSched. PID Parameters | linear interpolation in between*)
	tCtr_CDSu_In.Y_min_cust		:= -1.0;	(*"customized" Y-Min at the current moment (The existing Y-Min parameter is the global minimum. To have an effect Y_min_cust needs to be > the parameter | -1.0 = function not used*)
	tCtr_CDSu_In.Y_max_cust		:= 1.0;		(*"customized" Y-Max at the current moment (The existing Y-Max parameter is the global maximum. To have an effect Y_max_cust needs to be < the parameter | 1.0 = function not used*)
	tCtr_CDSu_In.Retrigger		:= FALSE;	(*a rising edge on this input signals the controller to retrigger - set W on X and force the Integrator to the current Y*)

	(* Input from Visualization via OPC *)
	tCtr_CDSu_In.Y_man_Active;
	tCtr_CDSu_In.Y_man;
	tCtr_CDSu_In.X_min;
	tCtr_CDSu_In.X_max;
	tCtr_CDSu_In.Tune_quality;
	tCtr_CDSu_In.Tune_PI;
	tCtr_CDSu_In.Tune_PID;
	tCtr_CDSu_In.Tune_start;
	tCtr_CDSu_In.Tune_stop;
	tCtr_CDSu_In.Tune_takeover;

	xCtr_CDSu();

	(* Output variables function block *)
	(* Output to module(s) *)
	OUT_HC.tCtr_CDSu_Set.Ao 	:= tCtr_CDSu_Out.Y;	(* analog out *)

	(* Output to Visualization via OPC *)
	MM2VIS.tCtr_CDSu_Out		:= tCtr_CDSu_Out;
	VIS2MM.tCtr_CDSu_In			:= tCtr_CDSu_In;	(* write back to IN_struct for reset: Tune_takeover, X-display, ...!*)

	tCtr_CDSu_Out.Active;
	tCtr_CDSu_Out.Y;
	tCtr_CDSu_Out.W;
	tCtr_CDSu_Out.e;
	tCtr_CDSu_Out.Kp_tune;
	tCtr_CDSu_Out.Tn_tune;
	tCtr_CDSu_Out.Tv_tune;
	tCtr_CDSu_Out.status;

END_PROGRAM
```

#### Ctr_CDSuInit.st
```iecst
PROGRAM _INIT

	xCtr_CDSu.pParameter := ADR(Para.tCtr_CDSu);
	xCtr_CDSu.pInput 	 := ADR(tCtr_CDSu_In);
	xCtr_CDSu.pOutput	 := ADR(tCtr_CDSu_Out);

	tCtr_CDSu_In.AlwaysUseYRamp		:= TRUE;	(*If TRUE the Y signal will always limit the change rate via the according parameter | if FALSE the Y signal will jump in case the controller is disabled (blocked or set)*)
	tCtr_CDSu_In.KeepYManAtBlock	:= TRUE;	(*If TRUE the controller will keep the Y-man value constant in case the controller is disabled (blocked or set) | If FALSE the blocked or set value will override the Y-man value*)
	tCtr_CDSu_In.Y_min_cust			:= -1.0;	(*"customized" Y-Min at the current moment (The existing Y-Min parameter is the global minimum. To have an effect Y_min_cust needs to be > the parameter | -1.0 = function not used*)
	tCtr_CDSu_In.Y_max_cust			:=  1.0;	(*"customized" Y-Max at the current moment (The existing Y-Max parameter is the global maximum. To have an effect Y_max_cust needs to be < the parameter | 1.0 = function not used*)
	tCtr_CDSu_In.StepperMode		:= FALSE;	(* TRUE = use PWM-Mode (standard mode until 4.10) | FALSE = use continuous servo drive *)

END_PROGRAM
```

### Program Logical/HeatingCooling/Ctr_ChC (IEC, version 4.12.0) - controller charge temperature

#### Ctr_ChCCyclic.st
```iecst
(*******************************************************************************
Ctr_ChC		charge temperature (cooler)

This code is confidential and proprietary to the INNIO Company.
It may not be used in any form, or reproduced in any manner,
without the express written permission of the INNIO Company.
Copyright, INNIO Company, 2022

Customized modifications: -
------------------------

History:
-------
V0.00.0		17.04.2012	lettenb.	created
V3.99.0		23.11.2012	lettenb.	write back to IN_struct added (zengerer)
V4.00.0		15.12.2014	lettenb.	controller interfaces completed like standard
V4.03.0     05.08.2015  Stary		added actual position feedback for regulator valve
V4.04.0		16.01.2017	lettenb.	demand CHC with bN_EngStart(request service eder andreas)
			11.05.2017	lettenb.	freeze ctr in case of bAMM_T_Ch_T2s_Avg(MS), SWAT920/2
V4.05.00.00	25.10.2017	Zengerer	rT_ChC_Ctr_Wex_Cust add V4.5 new interface
V4.05.01.00 25.03.2019	Fahringer	restart the controller to initiate the setpoint ramp
V4.11.00.00	28.01.2022	Perktold	included plant controller upgrade
V4.12.00.00	14.12.2022	Perktold	retrigger caused by X >= WMin just once per controller activation

Instructions for use:
--------------------

Outstandings:
------------
*******************************************************************************)

PROGRAM _CYCLIC

	(* Parameter *)
	Para.tCtr_ChC.W_set;
	Para.tCtr_ChC.W_set2;
	Para.tCtr_ChC.W_min;
	Para.tCtr_ChC.W_max;
	Para.tCtr_ChC.dW_up;
	Para.tCtr_ChC.dW_down;
	Para.tCtr_ChC.deadband;
	Para.tCtr_ChC.Y_min;
	Para.tCtr_ChC.Y_max;
	Para.tCtr_ChC.dY_max;
	Para.tCtr_ChC.Y_block;
	Para.tCtr_ChC.invert;
	Para.tCtr_ChC.Kp;
	Para.tCtr_ChC.Tn;
	Para.tCtr_ChC.Tv;
	Para.tCtr_ChC.Kp_GainScheduling;
	Para.tCtr_ChC.Tn_GainScheduling;
	Para.tCtr_ChC.Tv_GainScheduling;
	Para.tCtr_ChC.t_min_pulse_down;
	Para.tCtr_ChC.t_min_pulse_up;
	Para.tCtr_ChC.t_period_down;
	Para.tCtr_ChC.t_period_up;

	(* Input variables *)
	tCtr_ChC_In					:= VIS2MM.tCtr_ChC_In;		(* from vis *)

	(* Input from module *)
	tCtr_ChC_In.enable			:=	Para.bCtr_ChC
								AND	IN_HC.tPB2MM.bParaSetupOk
								AND IN_HC.bEng_Aux_Dem_CDR
								AND(bN_EngStart OR tCtr_ChC_In.enable);

	tCtr_ChC_In.W_ext_Active	:= VIS2MM.tCtr_ChC_In.W_ext_Active OR TRUE;

	IF IN_HC.bT_ChC_Ctr_Wex_Enable_Cust THEN							(*new V4.5*)
		tCtr_ChC_In.W_ext			:= IN_HC.rT_ChC_Ctr_Wex_Cust;
	ELSE
		tCtr_ChC_In.W_ext			:= IN_HC.rT_ChC_Ctr_Wex;
	END_IF

	tCtr_ChC_In.Y_set_Active	:= IN_HC.bAMM_T_Ch_T2s_Avg;//FALSE;	  freeze SWAT920/2
	tCtr_ChC_In.Y_set			:= 0.5;//0.0;	         			  freeze SWAT920/2
	tCtr_ChC_In.X				:= IN_HC.rT_Ch_T2s_Avg;
	tCtr_ChC_In.A				:= 0;
	tCtr_ChC_In.W_set2_Active	:= FALSE;	(*Input to define which internal setpoint will be used TRUE = use the 2nd set point | FALSE use the normal "1st" one*)
	tCtr_ChC_In.GainScheduling	:= 0.0;		(*Input for Gain Scheduling: 0.0 = use 100% of the Standard PID-Parameters | 1.0 = use 100% of the GainSched. PID Parameters | linear interpolation in between*)
	tCtr_ChC_In.Y_min_cust		:= -1.0;	(*"customized" Y-Min at the current moment (The existing Y-Min parameter is the global minimum. To have an effect Y_min_cust needs to be > the parameter | -1.0 = function not used*)
	tCtr_ChC_In.Y_max_cust		:= 1.0;		(*"customized" Y-Max at the current moment (The existing Y-Max parameter is the global maximum. To have an effect Y_max_cust needs to be < the parameter | 1.0 = function not used*)

	(* retrigger controller when Ctrl.X reached the minimum set point W_min and GCB is closed  OR closure of GCB*)
	tCtr_ChC_In.Retrigger := (EDGEPOS(tCtr_ChC_In.X >= Para.tCtr_ChC.W_min) AND NOT bBlockRetrigger) OR EDGEPOS(IN_HC.tGCB_On.Di);

	(* block retrigger caused be X >= WMin after one execution until controller is disabled again *)
	IF tCtr_ChC_In.Retrigger AND EDGEPOS(tCtr_ChC_In.X >= Para.tCtr_ChC.W_min) THEN
		bBlockRetrigger	:= TRUE;
	ELSIF bBlockRetrigger AND NOT tCtr_ChC_In.enable THEN
		bBlockRetrigger	:= FALSE;
	END_IF;
	(* Input from Visualization via OPC *)
	tCtr_ChC_In.Y_man_Active;
	tCtr_ChC_In.Y_man;
	tCtr_ChC_In.X_min;
	tCtr_ChC_In.X_max;
	tCtr_ChC_In.Tune_quality;
	tCtr_ChC_In.Tune_PI;
	tCtr_ChC_In.Tune_PID;
	tCtr_ChC_In.Tune_start;
	tCtr_ChC_In.Tune_stop;
	tCtr_ChC_In.Tune_takeover;

	xCtr_ChC();

	(* Output variables function block *)
	(* Output to module(s) *)
	OUT_HC.tCtr_ChC_Set.Ao 		:= tCtr_ChC_Out.Y;			(* analog out *)

	(* Output to Visualization via OPC *)
	MM2VIS.tCtr_ChC_Out			:= tCtr_ChC_Out;
	MM2VIS.rPos_ChC_Valve     	:= IN_HC.tPos_ChC_Valve.Ai;
	VIS2MM.tCtr_ChC_In			:= tCtr_ChC_In;				(* write back to IN_struct for reset: Tune_takeover, X-display, ...!*)

	tCtr_ChC_Out.Active;
	tCtr_ChC_Out.Y;
	tCtr_ChC_Out.W;
	tCtr_ChC_Out.e;
	tCtr_ChC_Out.Kp_tune;
	tCtr_ChC_Out.Tn_tune;
	tCtr_ChC_Out.Tv_tune;
	tCtr_ChC_Out.status;

END_PROGRAM
```

#### Ctr_ChCInit.st
```iecst
PROGRAM _INIT

	xCtr_ChC.pParameter := ADR(Para.tCtr_ChC);
	xCtr_ChC.pInput 	:= ADR(tCtr_ChC_In);
	xCtr_ChC.pOutput	:= ADR(tCtr_ChC_Out);

	tCtr_ChC_In.AlwaysUseYRamp		:= TRUE;	(*If TRUE the Y signal will always limit the change rate via the according parameter | if FALSE the Y signal will jump in case the controller is disabled (blocked or set)*)
	tCtr_ChC_In.KeepYManAtBlock		:= TRUE;	(*If TRUE the controller will keep the Y-man value constant in case the controller is disabled (blocked or set) | If FALSE the blocked or set value will override the Y-man value*)
	tCtr_ChC_In.Y_min_cust			:= -1.0;	(*"customized" Y-Min at the current moment (The existing Y-Min parameter is the global minimum. To have an effect Y_min_cust needs to be > the parameter | -1.0 = function not used*)
	tCtr_ChC_In.Y_max_cust			:=  1.0;	(*"customized" Y-Max at the current moment (The existing Y-Max parameter is the global maximum. To have an effect Y_max_cust needs to be < the parameter | 1.0 = function not used*)
	tCtr_ChC_In.StepperMode			:= FALSE;	(* TRUE = use PWM-Mode (standard mode until 4.10) | FALSE = use continuous servo drive *)

END_PROGRAM
```

#### Ctr_ChC.var
```iecst
(********************************************************************
 * COPYRIGHT -- INNIO Company
 ********************************************************************
 * Program: Ctr_ChC
 * File: Ctr_ChC.var
 * Author: lettenb
 * Created: April 17, 2012
 ********************************************************************
 * Local variables of program Ctr_ChC
 ********************************************************************)
VAR
	bBlockRetrigger : BOOL; (*block retrigger events*)
END_VAR
```

### Program Logical/HeatingCooling/Ctr_ChC_T1HP (IEC, version 4.11.0) - controller charge temperature before high-pressure turbo charger (T1-HP)

#### Ctr_ChC_T1HPCyclic.st
```iecst
(*******************************************************************************
Ctr_ChC_T1HP	charge temperature before high-pressure turbo charger (cooler)

This code is confidential and proprietary to the INNIO Company.
It may not be used in any form, or reproduced in any manner,
without the express written permission of the INNIO Company.
Copyright, INNIO Company, 2022

Customized modifications: -
------------------------

History:
-------
V0.00.0		09.08.2018	Schmid		created
V4.07.0		09.08.2018	Schmid		copy of Ctr_ChC, adapted to control T1-HP
			05.10.2018	Schmid		parameter OF ctr struct used FOR setpoint W_set (removed separate parameter)
V4.11.0		28.01.2022	Perktold	included plant controller upgrade

Instructions for use:
--------------------

Outstandings:
------------
*******************************************************************************)

PROGRAM _CYCLIC

	(* Parameter *)
	Para.tCtr_ChC_T1HP.W_set;
	Para.tCtr_ChC_T1HP.W_set2;
	Para.tCtr_ChC_T1HP.W_min;
	Para.tCtr_ChC_T1HP.W_max;
	Para.tCtr_ChC_T1HP.dW_up;
	Para.tCtr_ChC_T1HP.dW_down;
	Para.tCtr_ChC_T1HP.deadband;
	Para.tCtr_ChC_T1HP.Y_min;
	Para.tCtr_ChC_T1HP.Y_max;
	Para.tCtr_ChC_T1HP.dY_max;
	Para.tCtr_ChC_T1HP.Y_block;
	Para.tCtr_ChC_T1HP.invert;
	Para.tCtr_ChC_T1HP.Kp;
	Para.tCtr_ChC_T1HP.Tn;
	Para.tCtr_ChC_T1HP.Tv;
	Para.tCtr_ChC_T1HP.Kp_GainScheduling;
	Para.tCtr_ChC_T1HP.Tn_GainScheduling;
	Para.tCtr_ChC_T1HP.Tv_GainScheduling;
	Para.tCtr_ChC_T1HP.t_min_pulse_down;
	Para.tCtr_ChC_T1HP.t_min_pulse_up;
	Para.tCtr_ChC_T1HP.t_period_down;
	Para.tCtr_ChC_T1HP.t_period_up;

	(* Input variables *)
	tCtr_ChC_T1HP_In			:= VIS2MM.tCtr_ChC_T1HP_In;		(* from vis *)

	(* Input from module *)
	tCtr_ChC_T1HP_In.enable			:=	Para.bCtr_ChC_T1HP
									AND	IN_HC.tPB2MM.bParaSetupOk
									AND IN_HC.bEng_Aux_Dem_CDR
									AND(bN_EngStart OR tCtr_ChC_T1HP_In.enable);
	tCtr_ChC_T1HP_In.W_ext_Active	:= VIS2MM.tCtr_ChC_T1HP_In.W_ext_Active OR TRUE;
	tCtr_ChC_T1HP_In.W_ext			:= Para.tCtr_ChC_T1HP.W_set;
	tCtr_ChC_T1HP_In.Y_set_Active	:= IN_HC.bAMM_T_Ch_T1HP_Avg;//FALSE;	  freeze SWAT920/2
	tCtr_ChC_T1HP_In.Y_set			:= 0.5;//0.0;		         			  freeze SWAT920/2
	tCtr_ChC_T1HP_In.X				:= IN_HC.rT_Ch_T1HP_Avg;
	tCtr_ChC_T1HP_In.A				:= 0;
	tCtr_ChC_T1HP_In.W_set2_Active	:= FALSE;	(*Input to define which internal setpoint will be used TRUE = use the 2nd set point | FALSE use the normal "1st" one*)
	tCtr_ChC_T1HP_In.GainScheduling	:= 0.0;		(*Input for Gain Scheduling: 0.0 = use 100% of the Standard PID-Parameters | 1.0 = use 100% of the GainSched. PID Parameters | linear interpolation in between*)
	tCtr_ChC_T1HP_In.Y_min_cust		:= -1.0;	(*"customized" Y-Min at the current moment (The existing Y-Min parameter is the global minimum. To have an effect Y_min_cust needs to be > the parameter | -1.0 = function not used*)
	tCtr_ChC_T1HP_In.Y_max_cust		:= 1.0;		(*"customized" Y-Max at the current moment (The existing Y-Max parameter is the global maximum. To have an effect Y_max_cust needs to be < the parameter | 1.0 = function not used*)
	tCtr_ChC_T1HP_In.Retrigger		:= FALSE;	(*a rising edge on this input signals the controller to retrigger - set W on X and force the Integrator to the current Y*)

	(* Input from Visualization via OPC *)
	tCtr_ChC_T1HP_In.Y_man_Active;
	tCtr_ChC_T1HP_In.Y_man;
	tCtr_ChC_T1HP_In.X_min;
	tCtr_ChC_T1HP_In.X_max;
	tCtr_ChC_T1HP_In.Tune_quality;
	tCtr_ChC_T1HP_In.Tune_PI;
	tCtr_ChC_T1HP_In.Tune_PID;
	tCtr_ChC_T1HP_In.Tune_start;
	tCtr_ChC_T1HP_In.Tune_stop;
	tCtr_ChC_T1HP_In.Tune_takeover;

	xCtr_ChC_T1HP();

	(* Output variables function block *)
	(* Output to module(s) *)
	OUT_HC.tCtr_ChC2_Valve_Set.Ao	:= tCtr_ChC_T1HP_Out.Y;			(* analog out *)

	(* Output to Visualization via OPC *)
	MM2VIS.tCtr_ChC_T1HP_Out	:= tCtr_ChC_T1HP_Out;
	MM2VIS.rPos_ChC2_Valve		:= IN_HC.tPos_ChC2_Valve.Ai;
	VIS2MM.tCtr_ChC_T1HP_In		:= tCtr_ChC_T1HP_In;				(* write back to IN_struct for reset: Tune_takeover, X-display, ...!*)

	tCtr_ChC_T1HP_Out.Active;
	tCtr_ChC_T1HP_Out.Y;
	tCtr_ChC_T1HP_Out.W;
	tCtr_ChC_T1HP_Out.e;
	tCtr_ChC_T1HP_Out.Kp_tune;
	tCtr_ChC_T1HP_Out.Tn_tune;
	tCtr_ChC_T1HP_Out.Tv_tune;
	tCtr_ChC_T1HP_Out.status;

END_PROGRAM
```

#### Ctr_ChC_T1HPInit.st
```iecst
PROGRAM _INIT

	xCtr_ChC_T1HP.pParameter := ADR(Para.tCtr_ChC_T1HP);
	xCtr_ChC_T1HP.pInput 	:= ADR(tCtr_ChC_T1HP_In);
	xCtr_ChC_T1HP.pOutput	:= ADR(tCtr_ChC_T1HP_Out);

	tCtr_ChC_T1HP_In.AlwaysUseYRamp		:= TRUE;	(*If TRUE the Y signal will always limit the change rate via the according parameter | if FALSE the Y signal will jump in case the controller is disabled (blocked or set)*)
	tCtr_ChC_T1HP_In.KeepYManAtBlock	:= TRUE;	(*If TRUE the controller will keep the Y-man value constant in case the controller is disabled (blocked or set) | If FALSE the blocked or set value will override the Y-man value*)
	tCtr_ChC_T1HP_In.Y_min_cust			:= -1.0;	(*"customized" Y-Min at the current moment (The existing Y-Min parameter is the global minimum. To have an effect Y_min_cust needs to be > the parameter | -1.0 = function not used*)
	tCtr_ChC_T1HP_In.Y_max_cust			:=  1.0;	(*"customized" Y-Max at the current moment (The existing Y-Max parameter is the global maximum. To have an effect Y_max_cust needs to be < the parameter | 1.0 = function not used*)
	tCtr_ChC_T1HP_In.StepperMode		:= FALSE;	(* TRUE = use PWM-Mode (standard mode until 4.10) | FALSE = use continuous servo drive *)

END_PROGRAM
```

### Program Logical/HeatingCooling/Ctr_ChCV (IEC, version 4.11.0) - controller charge temperature cooler ventilation

#### Ctr_ChCVCyclic.st
```iecst
(*******************************************************************************
Ctr_ChCV		charge temperature cooler ventilation

This code is confidential and proprietary to the INNIO Company.
It may not be used in any form, or reproduced in any manner,
without the express written permission of the INNIO Company.
Copyright, INNIO Company, 2022

Customized modifications: -
------------------------

History:
-------
V0.00.0		17.04.2012	lettenb.	Created
V3.90.0		23.11.2012	lettenb.	write back to IN_struct added (zengerer)
V3.99.0		21.02.2013	lettenb.	IN_HC.tChCV_DemExt.Di (V3.30)
V4.00.0		15.12.2014	lettenb.	controller interfaces completed like standard
V4.11.0		28.01.2022	Perktold	included plant controller upgrade

Instructions for use:
--------------------

Outstandings:
------------
(*******************************************************************************)

PROGRAM _CYCLIC

	(* Parameter *)
	Para.tCtr_ChCV.W_set;
	Para.tCtr_ChCV.W_set2;
	Para.tCtr_ChCV.W_min;
	Para.tCtr_ChCV.W_max;
	Para.tCtr_ChCV.dW_up;
	Para.tCtr_ChCV.dW_down;
	Para.tCtr_ChCV.deadband;
	Para.tCtr_ChCV.Y_min;
	Para.tCtr_ChCV.Y_max;
	Para.tCtr_ChCV.dY_max;
	Para.tCtr_ChCV.Y_block;
	Para.tCtr_ChCV.invert;
	Para.tCtr_ChCV.Kp;
	Para.tCtr_ChCV.Tn;
	Para.tCtr_ChCV.Tv;
	Para.tCtr_ChCV.Kp_GainScheduling;
	Para.tCtr_ChCV.Tn_GainScheduling;
	Para.tCtr_ChCV.Tv_GainScheduling;
	Para.tCtr_ChCV.t_min_pulse_down;
	Para.tCtr_ChCV.t_min_pulse_up;
	Para.tCtr_ChCV.t_period_down;
	Para.tCtr_ChCV.t_period_up;

	(* Input variables *)
	tCtr_ChCV_In				:= VIS2MM.tCtr_ChCV_In;			(* from vis *)

	(* Input from module *)
	tCtr_ChCV_In.enable			:=	Para.bCtr_ChCV
								AND	IN_HC.tPB2MM.bParaSetupOk
								AND IN_HC.bEng_Aux_Dem_CDR;
	tCtr_ChCV_In.W_ext_Active	:= tCtr_ChCV_In.W_ext_Active OR TRUE;	(* from vis *)
	tCtr_ChCV_In.W_ext			:= Para.tCtr_ChCV.W_set - ((Para.rT_T2_Set[1] - IN_HC.rT_ChC_Ctr_Wex) * rChCV_Wex_factor);
	tCtr_ChCV_In.Y_set_Active	:= FALSE;
	tCtr_ChCV_In.Y_set			:= 0.0;
	tCtr_ChCV_In.X				:= IN_HC.rT_Ch_T2s_Avg;
	tCtr_ChCV_In.A				:= 0;
	tCtr_ChCV_In.W_set2_Active	:= FALSE;	(*Input to define which internal setpoint will be used TRUE = use the 2nd set point | FALSE use the normal "1st" one*)
	tCtr_ChCV_In.GainScheduling	:= 0.0;		(*Input for Gain Scheduling: 0.0 = use 100% of the Standard PID-Parameters | 1.0 = use 100% of the GainSched. PID Parameters | linear interpolation in between*)
	tCtr_ChCV_In.Y_min_cust		:= -1.0;	(*"customized" Y-Min at the current moment (The existing Y-Min parameter is the global minimum. To have an effect Y_min_cust needs to be > the parameter | -1.0 = function not used*)
	tCtr_ChCV_In.Y_max_cust		:= 1.0;		(*"customized" Y-Max at the current moment (The existing Y-Max parameter is the global maximum. To have an effect Y_max_cust needs to be < the parameter | 1.0 = function not used*)
	tCtr_ChCV_In.Retrigger		:= FALSE;	(*a rising edge on this input signals the controller to retrigger - set W on X and force the Integrator to the current Y*)

	(* Input from Visualization via OPC *)
	tCtr_ChCV_In.Y_man_Active;
	tCtr_ChCV_In.Y_man;
	tCtr_ChCV_In.X_min;
	tCtr_ChCV_In.X_max;
	tCtr_ChCV_In.Tune_quality;
	tCtr_ChCV_In.Tune_PI;
	tCtr_ChCV_In.Tune_PID;
	tCtr_ChCV_In.Tune_start;
	tCtr_ChCV_In.Tune_stop;
	tCtr_ChCV_In.Tune_takeover;

	xCtr_ChCV();

	(* Output variables function block *)
	(* Output to module(s) *)
	OUT_HC.tCtr_ChCV_Set.Ao 	:= tCtr_ChCV_Out.Y;		(* analog out *)

	(* Output to Visualization via OPC *)
	MM2VIS.tCtr_ChCV_Out		:= tCtr_ChCV_Out;
	VIS2MM.tCtr_ChCV_In			:= tCtr_ChCV_In;		(* write back to IN_struct for reset: Tune_takeover, X-display, ...!*)

	tCtr_ChCV_Out.Active;
	tCtr_ChCV_Out.Y;
	tCtr_ChCV_Out.W;
	tCtr_ChCV_Out.e;
	tCtr_ChCV_Out.Kp_tune;
	tCtr_ChCV_Out.Tn_tune;
	tCtr_ChCV_Out.Tv_tune;
	tCtr_ChCV_Out.status;

END_PROGRAM
```

#### Ctr_ChCVInit.st
```iecst
PROGRAM _INIT

	xCtr_ChCV.pParameter := ADR(Para.tCtr_ChCV);
	xCtr_ChCV.pInput  	 := ADR(tCtr_ChCV_In);
	xCtr_ChCV.pOutput	 := ADR(tCtr_ChCV_Out);

	tCtr_ChCV_In.AlwaysUseYRamp		:= TRUE;	(*If TRUE the Y signal will always limit the change rate via the according parameter | if FALSE the Y signal will jump in case the controller is disabled (blocked or set)*)
	tCtr_ChCV_In.KeepYManAtBlock	:= TRUE;	(*If TRUE the controller will keep the Y-man value constant in case the controller is disabled (blocked or set) | If FALSE the blocked or set value will override the Y-man value*)
	tCtr_ChCV_In.Y_min_cust			:= -1.0;	(*"customized" Y-Min at the current moment (The existing Y-Min parameter is the global minimum. To have an effect Y_min_cust needs to be > the parameter | -1.0 = function not used*)
	tCtr_ChCV_In.Y_max_cust			:=  1.0;	(*"customized" Y-Max at the current moment (The existing Y-Max parameter is the global maximum. To have an effect Y_max_cust needs to be < the parameter | 1.0 = function not used*)
	tCtr_ChCV_In.StepperMode		:= FALSE;	(* TRUE = use PWM-Mode (standard mode until 4.10) | FALSE = use continuous servo drive *)

END_PROGRAM
```

#### Ctr_ChCV.var
```iecst
VAR
	rChCV_Wex_factor : REAL := 1.0; (*charge cooler ventilation ctr Wex factor []*)
END_VAR
```

### Program Logical/HeatingCooling/Ctr_ChCHP (IEC, version 4.11.0) - controller charge temperature high pressure 

#### Ctr_ChCHPCyclic.st
```iecst
(*******************************************************************************
Ctr_ChCHP		charge temperature cooler high pressure

This code is confidential and proprietary to the INNIO Company.
It may not be used in any form, or reproduced in any manner,
without the express written permission of the INNIO Company.
Copyright, INNIO Company, 2022

Customized modifications: -
------------------------

History:
-------
V0.00.0		17.04.2012	lettenb.	Created
V3.99.0		23.11.2012	lettenb.	write back to IN_struct added (zengerer)
V4.00.0		15.12.2014	lettenb.	controller interfaces completed like standard
V4.11.0		28.01.2022	Perktold	included plant controller upgrade

Instructions for use:
--------------------

Outstandings:
------------
(*******************************************************************************)

PROGRAM _CYCLIC

	(* Parameter *)
	Para.tCtr_ChCHP.W_set;
	Para.tCtr_ChCHP.W_set2;
	Para.tCtr_ChCHP.W_min;
	Para.tCtr_ChCHP.W_max;
	Para.tCtr_ChCHP.dW_up;
	Para.tCtr_ChCHP.dW_down;
	Para.tCtr_ChCHP.deadband;
	Para.tCtr_ChCHP.Y_min;
	Para.tCtr_ChCHP.Y_max;
	Para.tCtr_ChCHP.dY_max;
	Para.tCtr_ChCHP.Y_block;
	Para.tCtr_ChCHP.invert;
	Para.tCtr_ChCHP.Kp;
	Para.tCtr_ChCHP.Tn;
	Para.tCtr_ChCHP.Tv;
	Para.tCtr_ChCHP.Kp_GainScheduling;
	Para.tCtr_ChCHP.Tn_GainScheduling;
	Para.tCtr_ChCHP.Tv_GainScheduling;
	Para.tCtr_ChCHP.t_min_pulse_down;
	Para.tCtr_ChCHP.t_min_pulse_up;
	Para.tCtr_ChCHP.t_period_down;
	Para.tCtr_ChCHP.t_period_up;

	(* Input variables *)
	tCtr_ChCHP_In				:= VIS2MM.tCtr_ChCHP_In;		(* from vis *)

	(* Input from module *)
	tCtr_ChCHP_In.enable		:=	Para.bCtr_ChCHP
								AND	IN_HC.tPB2MM.bParaSetupOk
								AND(IN_HC.bEng_Aux_Dem_CDR OR bN_EngStart);
	tCtr_ChCHP_In.W_ext_Active	:= tCtr_ChCHP_In.W_ext_Active;	(* from vis *)
	tCtr_ChCHP_In.W_ext			:= 0.0;
	tCtr_ChCHP_In.Y_set_Active	:= FALSE;
	tCtr_ChCHP_In.Y_set			:= 0.0;
	tCtr_ChCHP_In.X				:= IN_HC.rT_Ch_T2s_Avg;
	tCtr_ChCHP_In.A				:= 0;
	tCtr_ChCHP_In.W_set2_Active	:= FALSE;	(*Input to define which internal setpoint will be used TRUE = use the 2nd set point | FALSE use the normal "1st" one*)
	tCtr_ChCHP_In.GainScheduling:= 0.0;		(*Input for Gain Scheduling: 0.0 = use 100% of the Standard PID-Parameters | 1.0 = use 100% of the GainSched. PID Parameters | linear interpolation in between*)
	tCtr_ChCHP_In.Y_min_cust	:= -1.0;	(*"customized" Y-Min at the current moment (The existing Y-Min parameter is the global minimum. To have an effect Y_min_cust needs to be > the parameter | -1.0 = function not used*)
	tCtr_ChCHP_In.Y_max_cust	:= 1.0;		(*"customized" Y-Max at the current moment (The existing Y-Max parameter is the global maximum. To have an effect Y_max_cust needs to be < the parameter | 1.0 = function not used*)
	tCtr_ChCHP_In.Retrigger		:= FALSE;	(*a rising edge on this input signals the controller to retrigger - set W on X and force the Integrator to the current Y*)

	(* Input from Visualization via OPC *)
	tCtr_ChCHP_In.Y_man_Active;
	tCtr_ChCHP_In.Y_man;
	tCtr_ChCHP_In.X_min;
	tCtr_ChCHP_In.X_max;
	tCtr_ChCHP_In.Tune_quality;
	tCtr_ChCHP_In.Tune_PI;
	tCtr_ChCHP_In.Tune_PID;
	tCtr_ChCHP_In.Tune_start;
	tCtr_ChCHP_In.Tune_stop;
	tCtr_ChCHP_In.Tune_takeover;

	xCtr_ChCHP();

	(* Output variables function block *)
	(* Output to module(s) *)
	OUT_HC.tCtr_ChCHP_Set.Ao 	:= tCtr_ChCHP_Out.Y;	(* analog out *)

	(* Output to Visualization via OPC *)
	MM2VIS.tCtr_ChCHP_Out		:= tCtr_ChCHP_Out;
	VIS2MM.tCtr_ChCHP_In		:= tCtr_ChCHP_In;		(* write back to IN_struct for reset: Tune_takeover, X-display, ...!*)

	tCtr_ChCHP_Out.Active;
	tCtr_ChCHP_Out.Y;
	tCtr_ChCHP_Out.W;
	tCtr_ChCHP_Out.e;
	tCtr_ChCHP_Out.Kp_tune;
	tCtr_ChCHP_Out.Tn_tune;
	tCtr_ChCHP_Out.Tv_tune;
	tCtr_ChCHP_Out.status;

END_PROGRAM
```

#### Ctr_ChCHPInit.st
```iecst
PROGRAM _INIT

	xCtr_ChCHP.pParameter := ADR(Para.tCtr_ChCHP);
	xCtr_ChCHP.pInput 	  := ADR(tCtr_ChCHP_In);
	xCtr_ChCHP.pOutput	  := ADR(tCtr_ChCHP_Out);

	tCtr_ChCHP_In.AlwaysUseYRamp		:= TRUE;	(*If TRUE the Y signal will always limit the change rate via the according parameter | if FALSE the Y signal will jump in case the controller is disabled (blocked or set)*)
	tCtr_ChCHP_In.KeepYManAtBlock		:= TRUE;	(*If TRUE the controller will keep the Y-man value constant in case the controller is disabled (blocked or set) | If FALSE the blocked or set value will override the Y-man value*)
	tCtr_ChCHP_In.Y_min_cust			:= -1.0;	(*"customized" Y-Min at the current moment (The existing Y-Min parameter is the global minimum. To have an effect Y_min_cust needs to be > the parameter | -1.0 = function not used*)
	tCtr_ChCHP_In.Y_max_cust			:=  1.0;	(*"customized" Y-Max at the current moment (The existing Y-Max parameter is the global maximum. To have an effect Y_max_cust needs to be < the parameter | 1.0 = function not used*)
	tCtr_ChCHP_In.StepperMode			:= FALSE;	(* TRUE = use PWM-Mode (standard mode until 4.10) | FALSE = use continuous servo drive *)

END_PROGRAM
```

### Program Logical/HeatingCooling/Ctr_HWRe (IEC, version 4.12.0) - controller heat water return temperature

#### Ctr_HWReCyclic.st
```iecst
(*******************************************************************************
Ctr_HWRe		heat water return temperature

This code is confidential and proprietary to the INNIO Company.
It may not be used in any form, or reproduced in any manner,
without the express written permission of the INNIO Company.
Copyright, INNIO Company, 2022

Customized modifications: -
------------------------

History:
-------
V0.00.0		17.04.2012  lettenbichler	Created
V3.99.0		23.11.2012	lettenbichler	write back to IN_struct added (zengerer)
V4.00.0		15.12.2014	lettenb.		controller interfaces completed like standard
V4.03.0     05.08.2015  Stary			added actual position feedback for regulator valve
V4.04.0		28.09.2016	lettenb.		tCtr_HWRe_In.X writing depending on parameter (kluckner)
V4.04.1		03.04.2019	Fahringer		restart the controller to initiate the setpoint ramp
V4.11.0		28.01.2022	Perktold		included plant controller upgrade
V4.12.0		14.12.2022	Perktold		retrigger caused by X >= WMin just once per controller activation

Instructions for use:
--------------------

Outstandings:
------------
(*******************************************************************************)

PROGRAM _CYCLIC

	(* Parameter *)
	Para.tCtr_HWRe.W_set;
	Para.tCtr_HWRe.W_set2;
	Para.tCtr_HWRe.W_min;
	Para.tCtr_HWRe.W_max;
	Para.tCtr_HWRe.dW_up;
	Para.tCtr_HWRe.dW_down;
	Para.tCtr_HWRe.deadband;
	Para.tCtr_HWRe.Y_min;
	Para.tCtr_HWRe.Y_max;
	Para.tCtr_HWRe.dY_max;
	Para.tCtr_HWRe.Y_block;
	Para.tCtr_HWRe.invert;
	Para.tCtr_HWRe.Kp;
	Para.tCtr_HWRe.Tn;
	Para.tCtr_HWRe.Tv;
//	Para.tCtr_HWRe.Kp_manualAdjust;
//	Para.tCtr_HWRe.Tn_manualAdjust;
//	Para.tCtr_HWRe.Tv_manualAdjust;
	Para.tCtr_HWRe.t_min_pulse_down;
	Para.tCtr_HWRe.t_min_pulse_up;
	Para.tCtr_HWRe.t_period_down;
	Para.tCtr_HWRe.t_period_up;

	(* Input variables *)
	tCtr_HWRe_In				:= VIS2MM.tCtr_HWRe_In;			(* from vis *)

	(* Input from module *)
	tCtr_HWRe_In.enable			:=	Para.bCtr_HWRe
								AND IN_HC.tPB2MM.bParaSetupOk
								AND IN_HC.bEng_Aux_Dem_CDR;

	tCtr_HWRe_In.W_ext_Active	:= tCtr_HWRe_In.W_ext_Active;	(* from vis *)
	tCtr_HWRe_In.W_ext			:= 0.0;
	tCtr_HWRe_In.Y_set_Active	:= FALSE;
	tCtr_HWRe_In.Y_set			:= 0.0;
	IF Para.bT_HW_Re_Active THEN tCtr_HWRe_In.X	:= IN_HC.tT_HW_Re.Ai;
	ELSE						 tCtr_HWRe_In.X	:= IN_HC.tT_HW_ReBeEng.Ai;
	END_IF;
	tCtr_HWRe_In.A				:= 0;
	tCtr_HWRe_In.W_set2_Active	:= FALSE;	(*Input to define which internal setpoint will be used TRUE = use the 2nd set point | FALSE use the normal "1st" one*)
	tCtr_HWRe_In.GainScheduling	:= 0.0;		(*Input for Gain Scheduling: 0.0 = use 100% of the Standard PID-Parameters | 1.0 = use 100% of the GainSched. PID Parameters | linear interpolation in between*)
	tCtr_HWRe_In.Y_min_cust		:= -1.0;	(*"customized" Y-Min at the current moment (The existing Y-Min parameter is the global minimum. To have an effect Y_min_cust needs to be > the parameter | -1.0 = function not used*)
	tCtr_HWRe_In.Y_max_cust		:= 1.0;		(*"customized" Y-Max at the current moment (The existing Y-Max parameter is the global maximum. To have an effect Y_max_cust needs to be < the parameter | 1.0 = function not used*)

	(* retrigger controller when Ctrl.X reached the minimum set point W_min and GCB is closed  OR closure of GCB*)
	tCtr_HWRe_In.Retrigger := (EDGEPOS(tCtr_HWRe_In.X >= Para.tCtr_HWRe.W_min) AND NOT bBlockRetrigger) OR EDGEPOS(IN_HC.tGCB_On.Di);

	(* block retrigger caused be X >= WMin after one execution until controller is disabled again *)
	IF tCtr_HWRe_In.Retrigger AND EDGEPOS(tCtr_HWRe_In.X >= Para.tCtr_HWRe.W_min) THEN
		bBlockRetrigger	:= TRUE;
	ELSIF bBlockRetrigger AND NOT tCtr_HWRe_In.enable THEN
		bBlockRetrigger	:= FALSE;
	END_IF;

	(* Input from Visualization via OPC *)
	tCtr_HWRe_In.Y_man_Active;
	tCtr_HWRe_In.Y_man;
	tCtr_HWRe_In.X_min;
	tCtr_HWRe_In.X_max;
	tCtr_HWRe_In.Tune_quality;
	tCtr_HWRe_In.Tune_PI;
	tCtr_HWRe_In.Tune_PID;
	tCtr_HWRe_In.Tune_start;
	tCtr_HWRe_In.Tune_stop;
	tCtr_HWRe_In.Tune_takeover;

	xCtr_HWRe();

	(* Output variables function block *)
	(* Output to module(s) *)
	OUT_HC.tCtr_HWRe_Set.Ao 	:= tCtr_HWRe_Out.Y;		(* analog out *)

	(* Output to Visualization via OPC *)
	MM2VIS.tCtr_HWRe_Out		:= tCtr_HWRe_Out;
	MM2VIS.rPos_HW_ReValve      := IN_HC.tPos_HW_ReValve.Ai;
	VIS2MM.tCtr_HWRe_In			:= tCtr_HWRe_In;		(* write back to IN_struct for reset: Tune_takeover, X-display, ...!*)

	tCtr_HWRe_Out.Active;
	tCtr_HWRe_Out.Y;
	tCtr_HWRe_Out.W;
	tCtr_HWRe_Out.e;
	tCtr_HWRe_Out.Kp_tune;
	tCtr_HWRe_Out.Tn_tune;
	tCtr_HWRe_Out.Tv_tune;
	tCtr_HWRe_Out.status;

END_PROGRAM
```

#### Ctr_HWReInit.st
```iecst
PROGRAM _INIT

	xCtr_HWRe.pParameter := ADR(Para.tCtr_HWRe);
	xCtr_HWRe.pInput 	 := ADR(tCtr_HWRe_In);
	xCtr_HWRe.pOutput	 := ADR(tCtr_HWRe_Out);

	tCtr_HWRe_In.AlwaysUseYRamp		:= TRUE;	(*If TRUE the Y signal will always limit the change rate via the according parameter | if FALSE the Y signal will jump in case the controller is disabled (blocked or set)*)
	tCtr_HWRe_In.KeepYManAtBlock	:= TRUE;	(*If TRUE the controller will keep the Y-man value constant in case the controller is disabled (blocked or set) | If FALSE the blocked or set value will override the Y-man value*)
	tCtr_HWRe_In.Y_min_cust			:= -1.0;	(*"customized" Y-Min at the current moment (The existing Y-Min parameter is the global minimum. To have an effect Y_min_cust needs to be > the parameter | -1.0 = function not used*)
	tCtr_HWRe_In.Y_max_cust			:=  1.0;	(*"customized" Y-Max at the current moment (The existing Y-Max parameter is the global maximum. To have an effect Y_max_cust needs to be < the parameter | 1.0 = function not used*)
	tCtr_HWRe_In.StepperMode		:= FALSE;	(* TRUE = use PWM-Mode (standard mode until 4.10) | FALSE = use continuous servo drive *)

END_PROGRAM
```

#### Ctr_HWRe.var
```iecst
(********************************************************************
 * COPYRIGHT -- INNIO Company
 ********************************************************************
 * Program: Ctr_T_HW_Re
 * File: Ctr_T_HW_Re.var
 * Author: lettenb
 * Created: April 17, 2012
 ********************************************************************
 * Local variables of program Ctr_T_HW_Re
 ********************************************************************)
VAR
	bBlockRetrigger : BOOL; (*block retrigger events*)
END_VAR
```

### Program Logical/HeatingCooling/Ctr_EC (IEC, version 4.11.0) - controller heat water return temperature after emergency cooler

#### Ctr_ECCyclic.st
```iecst
(*******************************************************************************
Ctr_EC		controller heat water return temperature after emergency cooler

This code is confidential and proprietary to the INNIO Company.
It may not be used in any form, or reproduced in any manner,
without the express written permission of the INNIO Company.
Copyright, INNIO Company, 2022

Customized modifications: -
------------------------

History:
-------
V0.00.0		17.04.2012 	lettenb.	Created
V3.99.0		23.11.2012	lettenb.	write back to IN_struct added (zengerer)
V4.00.0		15.12.2014	lettenb.	controller interfaces completed like standard
V4.03.0     05.08.2015  Stary		added actual position feedback for regulator valve
V4.11.0		28.01.2022	Perktold	included plant controller upgrade

Instructions for use:
--------------------

Outstandings:
------------
(*******************************************************************************)

PROGRAM _CYCLIC

	(* Parameter *)
	Para.tCtr_EC.W_set;
	Para.tCtr_EC.W_set2;
	Para.tCtr_EC.W_min;
	Para.tCtr_EC.W_max;
	Para.tCtr_EC.dW_up;
	Para.tCtr_EC.dW_down;
	Para.tCtr_EC.deadband;
	Para.tCtr_EC.Y_min;
	Para.tCtr_EC.Y_max;
	Para.tCtr_EC.dY_max;
	Para.tCtr_EC.Y_block;
	Para.tCtr_EC.invert;
	Para.tCtr_EC.Kp;
	Para.tCtr_EC.Tn;
	Para.tCtr_EC.Tv;
	Para.tCtr_EC.Kp_GainScheduling;
	Para.tCtr_EC.Tn_GainScheduling;
	Para.tCtr_EC.Tv_GainScheduling;
	Para.tCtr_EC.t_min_pulse_down;
	Para.tCtr_EC.t_min_pulse_up;
	Para.tCtr_EC.t_period_down;
	Para.tCtr_EC.t_period_up;

	(* Input variables *)
	tCtr_EC_In					:= VIS2MM.tCtr_EC_In;		(* from vis *)

	(* Input from module *)
	tCtr_EC_In.enable			:=	Para.bCtr_EC
								AND IN_HC.tPB2MM.bParaSetupOk
								AND IN_HC.bEng_Aux_Dem_CDR;
	tCtr_EC_In.W_ext_Active		:= tCtr_EC_In.W_ext_Active;	(* from vis *)
	tCtr_EC_In.W_ext			:= 0.0;
	tCtr_EC_In.Y_set_Active		:= FALSE;
	tCtr_EC_In.Y_set			:= 0.0;
	tCtr_EC_In.X				:= IN_HC.tT_HW_ReAfEC.Ai;
	tCtr_EC_In.A				:= 0;
	tCtr_EC_In.W_set2_Active	:= FALSE;	(*Input to define which internal setpoint will be used TRUE = use the 2nd set point | FALSE use the normal "1st" one*)
	tCtr_EC_In.GainScheduling	:= 0.0;		(*Input for Gain Scheduling: 0.0 = use 100% of the Standard PID-Parameters | 1.0 = use 100% of the GainSched. PID Parameters | linear interpolation in between*)
	tCtr_EC_In.Y_min_cust		:= -1.0;	(*"customized" Y-Min at the current moment (The existing Y-Min parameter is the global minimum. To have an effect Y_min_cust needs to be > the parameter | -1.0 = function not used*)
	tCtr_EC_In.Y_max_cust		:= 1.0;		(*"customized" Y-Max at the current moment (The existing Y-Max parameter is the global maximum. To have an effect Y_max_cust needs to be < the parameter | 1.0 = function not used*)
	tCtr_EC_In.Retrigger		:= FALSE;	(*a rising edge on this input signals the controller to retrigger - set W on X and force the Integrator to the current Y*)

	(* Input from Visualization via OPC *)
	tCtr_EC_In.Y_man_Active;
	tCtr_EC_In.Y_man;
	tCtr_EC_In.X_min;
	tCtr_EC_In.X_max;
	tCtr_EC_In.Tune_quality;
	tCtr_EC_In.Tune_PI;
	tCtr_EC_In.Tune_PID;
	tCtr_EC_In.Tune_start;
	tCtr_EC_In.Tune_stop;
	tCtr_EC_In.Tune_takeover;

	xCtr_EC();

	(* Output variables function block *)
	(* Output to module(s) *)
	OUT_HC.tCtr_EC_Set.Ao 		:= tCtr_EC_Out.Y;	(* analog out *)

	(* Output to Visualization via OPC *)
	MM2VIS.tCtr_EC_Out			:= tCtr_EC_Out;
	MM2VIS.rPos_HW_EC_ReValve   := IN_HC.tPos_HW_EC_ReValve.Ai;
	VIS2MM.tCtr_EC_In			:= tCtr_EC_In;		(* write back to IN_struct for reset: Tune_takeover, X-display, ...!*)

	tCtr_EC_Out.Active;
	tCtr_EC_Out.Y;
	tCtr_EC_Out.W;
	tCtr_EC_Out.e;
	tCtr_EC_Out.Kp_tune;
	tCtr_EC_Out.Tn_tune;
	tCtr_EC_Out.Tv_tune;
	tCtr_EC_Out.status;

END_PROGRAM
```

#### Ctr_ECInit.st
```iecst
PROGRAM _INIT

	xCtr_EC.pParameter 	:= ADR(Para.tCtr_EC);
	xCtr_EC.pInput 		:= ADR(tCtr_EC_In);
	xCtr_EC.pOutput	 	:= ADR(tCtr_EC_Out);

	tCtr_EC_In.AlwaysUseYRamp		:= TRUE;	(*If TRUE the Y signal will always limit the change rate via the according parameter | if FALSE the Y signal will jump in case the controller is disabled (blocked or set)*)
	tCtr_EC_In.KeepYManAtBlock		:= TRUE;	(*If TRUE the controller will keep the Y-man value constant in case the controller is disabled (blocked or set) | If FALSE the blocked or set value will override the Y-man value*)
	tCtr_EC_In.Y_min_cust			:= -1.0;	(*"customized" Y-Min at the current moment (The existing Y-Min parameter is the global minimum. To have an effect Y_min_cust needs to be > the parameter | -1.0 = function not used*)
	tCtr_EC_In.Y_max_cust			:=  1.0;	(*"customized" Y-Max at the current moment (The existing Y-Max parameter is the global maximum. To have an effect Y_max_cust needs to be < the parameter | 1.0 = function not used*)
	tCtr_EC_In.StepperMode			:= FALSE;	(* TRUE = use PWM-Mode (standard mode until 4.10) | FALSE = use continuous servo drive *)

END_PROGRAM
```

### Program Logical/HeatingCooling/Ctr_HWSu (IEC, version 4.11.0) - controller heat water supply temperature
